# B&R Automation Studio project NAEUL004C00R13L518F00 (part 18)

#### Act_OptP0929MagConv2BtmDC.st
```iecst
ACTION Act_OptP0929MagConv2BtmDC:

	//Magazine Conv2eyor
	IF tyP0929MagConv2.tyBtmDC.tyBtnStop.bRtCompl = TRUE THEN
		eOutMagConv2Act	:= MagConvActStop;

		IF p_eOutMagConv2Stat = MagConvActStop AND p_eOutMagConv2Status = Done THEN
			eOutMagConv2Act	:= MagConvActIdle;

			tyP0929MagConv2.tyBtmDC.tyBtnStop.bRtCompl		:= FALSE;
			tyP0929MagConv2.tyBtmDC.tyBtnStop.bValue		:= TRUE;
			tyP0929MagConv2.tyBtmDC.tyBtnStop.bRtLk		:= TRUE;

			tyP0929MagConv2.tyBtmDC.tyBtnMagIn.bRtCompl	:= FALSE;
			tyP0929MagConv2.tyBtmDC.tyBtnMagIn.bValue		:= FALSE;
			tyP0929MagConv2.tyBtmDC.tyBtnMagIn.bRtLk		:= FALSE;

			tyP0929MagConv2.tyBtmDC.tyBtnMagOut.bRtCompl	:= FALSE;
			tyP0929MagConv2.tyBtmDC.tyBtnMagOut.bValue		:= FALSE;
			tyP0929MagConv2.tyBtmDC.tyBtnMagOut.bRtLk		:= FALSE;
		END_IF

	ELSIF tyP0929MagConv2.tyBtmDC.tyBtnMagIn.bRtCompl = TRUE THEN
		tyP0929MagConv2.tyBtmDC.tyBtnMagIn.bValue	:= TRUE;
		tyP0929MagConv2.tyBtmDC.tyBtnMagIn.bRtLk	:= TRUE;

		tyP0929MagConv2.tyBtmDC.tyBtnStop.bValue	:= FALSE;
		tyP0929MagConv2.tyBtmDC.tyBtnStop.bRtLk	:= FALSE;

		IF p_tyNtParamCurr.eProjOutMagConv2Dir = ConvDirLToR OR p_tyNtParamCurr.eProjOutMagConv2Dir = ConvDirLToL THEN

			eOutMagConv2Act	:= MagConvActSetMtrSigOnOrLToR;

			IF p_eOutMagConv2Stat = MagConvActSetMtrSigOnOrLToR AND p_eOutMagConv2Status = Done THEN
				eOutMagConv2Act	:= MagConvActIdle;

				tyP0929MagConv2.tyBtmDC.tyBtnMagIn.bRtCompl	:= FALSE;
			END_IF

		ELSE

			eOutMagConv2Act	:= MagConvActSetMtrDirOrRToL;

			IF p_eOutMagConv2Stat = MagConvActSetMtrDirOrRToL AND p_eOutMagConv2Status = Done THEN
				eOutMagConv2Act	:= MagConvActIdle;

				tyP0929MagConv2.tyBtmDC.tyBtnMagIn.bRtCompl	:= FALSE;
			END_IF

		END_IF

	ELSIF tyP0929MagConv2.tyBtmDC.tyBtnMagOut.bRtCompl = TRUE THEN
		tyP0929MagConv2.tyBtmDC.tyBtnMagOut.bValue	:= TRUE;
		tyP0929MagConv2.tyBtmDC.tyBtnMagOut.bRtLk	:= TRUE;

		tyP0929MagConv2.tyBtmDC.tyBtnStop.bValue	:= FALSE;
		tyP0929MagConv2.tyBtmDC.tyBtnStop.bRtLk	:= FALSE;

		IF p_tyNtParamCurr.eProjOutMagConv2Dir = ConvDirLToR OR p_tyNtParamCurr.eProjOutMagConv2Dir = ConvDirRToR THEN

			eOutMagConv2Act	:= MagConvActSetMtrSigOnOrLToR;

			IF p_eOutMagConv2Stat = MagConvActSetMtrSigOnOrLToR AND p_eOutMagConv2Status = Done THEN
				eOutMagConv2Act	:= MagConvActIdle;

				tyP0929MagConv2.tyBtmDC.tyBtnMagOut.bRtCompl	:= FALSE;
			END_IF

		ELSE

			eOutMagConv2Act	:= MagConvActSetMtrDirOrRToL;

			IF p_eOutMagConv2Stat = MagConvActSetMtrDirOrRToL AND p_eOutMagConv2Status = Done THEN
				eOutMagConv2Act	:= MagConvActIdle;

				tyP0929MagConv2.tyBtmDC.tyBtnMagOut.bRtCompl	:= FALSE;
			END_IF

		END_IF

	END_IF

	IF tyP0929MagConv2.tyCom.tyBtnSwitch.bValue = TRUE THEN

		//Mag Conv2 Stopper4
		IF p_bStopper4TwoCtrlOut = FALSE THEN
			IF tyP0929MagConv2.tyBtmDC.tyBtnMidStprExt.bRtCompl = TRUE THEN
				tyP0929MagConv2.tyBtmDC.tyBtnMidStprExt.bValue := TRUE;
				tyP0929MagConv2.tyBtmDC.tyBtnMidStprRet.bValue := FALSE;

				eStopper4Act2	:= PneuActSetExt;

				IF p_eStopper4Stat2 = PneuActSetExt AND p_eStopper4Status2 = Done THEN
					eStopper4Act2	:= PneuActIdle;

					tyP0929MagConv2.tyBtmDC.tyBtnMidStprExt.bRtCompl	:= FALSE;
				END_IF

			ELSIF tyP0929MagConv2.tyBtmDC.tyBtnMidStprRet.bRtCompl = TRUE THEN
				tyP0929MagConv2.tyBtmDC.tyBtnMidStprRet.bValue := TRUE;
				tyP0929MagConv2.tyBtmDC.tyBtnMidStprExt.bValue := FALSE;

				eStopper4Act2	:= PneuActSetRet;

				IF p_eStopper4Stat2 = PneuActSetRet AND p_eStopper4Status2 = Done THEN
					eStopper4Act2	:= PneuActIdle;

					tyP0929MagConv2.tyBtmDC.tyBtnMidStprRet.bRtCompl	:= FALSE;
				END_IF
			END_IF

		ELSE
			IF (tyP0929MagConv2.tyBtmDC.tyBtnMidStprExt.bRtCompl = TRUE) OR (tyP0929MagConv2.tyBtmDC.tyBtnMidStprRet.bRtCompl = TRUE) THEN
				IF (tyP0929MagConv2.tyBtmDC.tyBtnMidStprExt.bValue = TRUE) AND (tyP0929MagConv2.tyBtmDC.tyBtnMidStprRet.bValue = TRUE) THEN
					eStopper4Act2	:= PneuActSetAll;

					IF p_eStopper4Stat2 = PneuActSetAll AND p_eStopper4Status2 = Done THEN
						eStopper4Act2	:= PneuActIdle;

						tyP0929MagConv2.tyBtmDC.tyBtnMidStprExt.bRtCompl		:= FALSE;
						tyP0929MagConv2.tyBtmDC.tyBtnMidStprRet.bRtCompl			:= FALSE;
					END_IF
					/////////i edited the ret to ext
				ELSIF (tyP0929MagConv2.tyBtmDC.tyBtnMidStprExt.bValue = TRUE) AND (tyP0929MagConv2.tyBtmDC.tyBtnMidStprRet.bValue = FALSE) THEN
					eStopper4Act2	:= PneuActSetExt;(**)

					IF p_eStopper4Stat2 = PneuActSetExt (**) AND p_eStopper4Status2 = Done THEN
						eStopper4Act2	:= PneuActIdle;

						tyP0929MagConv2.tyBtmDC.tyBtnMidStprExt.bRtCompl		:= FALSE;
						tyP0929MagConv2.tyBtmDC.tyBtnMidStprRet.bRtCompl		:= FALSE;
					END_IF

				ELSIF (tyP0929MagConv2.tyBtmDC.tyBtnMidStprExt.bValue = FALSE) AND (tyP0929MagConv2.tyBtmDC.tyBtnMidStprRet.bValue = TRUE) THEN
					eStopper4Act2	:= PneuActSetRet;

					IF p_eStopper4Stat2 = PneuActSetRet AND p_eStopper4Status2 = Done THEN
						eStopper4Act2	:= PneuActIdle;

						tyP0929MagConv2.tyBtmDC.tyBtnMidStprExt.bRtCompl		:= FALSE;
						tyP0929MagConv2.tyBtmDC.tyBtnMidStprRet.bRtCompl			:= FALSE;
					END_IF
					///////
				ELSE
					eStopper4Act2	:= PneuActRstAll;

					IF p_eStopper4Stat2 = PneuActRstAll AND p_eStopper4Status2 = Done THEN
						eStopper4Act2	:= PneuActIdle;

						tyP0929MagConv2.tyBtmDC.tyBtnMidStprExt.bRtCompl		:= FALSE;
						tyP0929MagConv2.tyBtmDC.tyBtnMidStprRet.bRtCompl			:= FALSE;
					END_IF

				END_IF
			END_IF
		END_IF//Stopper4

		//Mag Conv2 Stopper5
		IF p_bStopper5TwoCtrlOut = FALSE THEN
			IF tyP0929MagConv2.tyBtmDC.tyBtnExtStprExt.bRtCompl = TRUE THEN
				tyP0929MagConv2.tyBtmDC.tyBtnExtStprExt.bValue := TRUE;
				tyP0929MagConv2.tyBtmDC.tyBtnExtStprRet.bValue := FALSE;

				eStopper5Act2	:= PneuActSetExt;

				IF p_eStopper5Stat2 = PneuActSetExt AND p_eStopper5Status2 = Done THEN
					eStopper5Act2	:= PneuActIdle;

					tyP0929MagConv2.tyBtmDC.tyBtnExtStprExt.bRtCompl	:= FALSE;
				END_IF

			ELSIF tyP0929MagConv2.tyBtmDC.tyBtnExtStprRet.bRtCompl = TRUE THEN
				tyP0929MagConv2.tyBtmDC.tyBtnExtStprRet.bValue := TRUE;
				tyP0929MagConv2.tyBtmDC.tyBtnExtStprExt.bValue := FALSE;

				eStopper5Act2	:= PneuActSetRet;

				IF p_eStopper5Stat2 = PneuActSetRet AND p_eStopper5Status2 = Done THEN
					eStopper5Act2	:= PneuActIdle;

					tyP0929MagConv2.tyBtmDC.tyBtnExtStprRet.bRtCompl	:= FALSE;
				END_IF
			END_IF

		ELSE
			IF (tyP0929MagConv2.tyBtmDC.tyBtnExtStprExt.bRtCompl = TRUE) OR (tyP0929MagConv2.tyBtmDC.tyBtnExtStprRet.bRtCompl = TRUE) THEN
				IF (tyP0929MagConv2.tyBtmDC.tyBtnExtStprExt.bValue = TRUE) AND (tyP0929MagConv2.tyBtmDC.tyBtnExtStprRet.bValue = TRUE) THEN
					eStopper5Act2	:= PneuActSetAll;

					IF p_eStopper5Stat2 = PneuActSetAll AND p_eStopper5Status2 = Done THEN
						eStopper5Act2	:= PneuActIdle;

						tyP0929MagConv2.tyBtmDC.tyBtnExtStprExt.bRtCompl		:= FALSE;
						tyP0929MagConv2.tyBtmDC.tyBtnExtStprRet.bRtCompl			:= FALSE;
					END_IF
					/////////i edited the ret to ext
				ELSIF (tyP0929MagConv2.tyBtmDC.tyBtnExtStprExt.bValue = TRUE) AND (tyP0929MagConv2.tyBtmDC.tyBtnExtStprRet.bValue = FALSE) THEN
					eStopper5Act2	:= PneuActSetExt;(**)

					IF p_eStopper5Stat2 = PneuActSetExt (**) AND p_eStopper5Status2 = Done THEN
						eStopper5Act2	:= PneuActIdle;

						tyP0929MagConv2.tyBtmDC.tyBtnExtStprExt.bRtCompl		:= FALSE;
						tyP0929MagConv2.tyBtmDC.tyBtnExtStprRet.bRtCompl		:= FALSE;
					END_IF

				ELSIF (tyP0929MagConv2.tyBtmDC.tyBtnExtStprExt.bValue = FALSE) AND (tyP0929MagConv2.tyBtmDC.tyBtnExtStprRet.bValue = TRUE) THEN
					eStopper5Act2	:= PneuActSetRet;

					IF p_eStopper5Stat2 = PneuActSetRet AND p_eStopper5Status2 = Done THEN
						eStopper5Act2	:= PneuActIdle;

						tyP0929MagConv2.tyBtmDC.tyBtnExtStprExt.bRtCompl		:= FALSE;
						tyP0929MagConv2.tyBtmDC.tyBtnExtStprRet.bRtCompl			:= FALSE;
					END_IF
					///////
				ELSE
					eStopper5Act2	:= PneuActRstAll;

					IF p_eStopper5Stat2 = PneuActRstAll AND p_eStopper5Status2 = Done THEN
						eStopper5Act2	:= PneuActIdle;

						tyP0929MagConv2.tyBtmDC.tyBtnExtStprExt.bRtCompl		:= FALSE;
						tyP0929MagConv2.tyBtmDC.tyBtnExtStprRet.bRtCompl			:= FALSE;
					END_IF

				END_IF
			END_IF
		END_IF//Stopper5

		//mid
		tyP0929MagConv2.tyBtmFB.tyBtnMidStprExt.bRtCompl		:= FALSE;
		tyP0929MagConv2.tyBtmFB.tyBtnMidStprExt.bValue		:= FALSE;
		tyP0929MagConv2.tyBtmFB.tyBtnMidStprRet.bRtCompl		:= FALSE;
		tyP0929MagConv2.tyBtmFB.tyBtnMidStprRet.bValue		:= FALSE;

		//ext
		tyP0929MagConv2.tyBtmFB.tyBtnExtStprExt.bRtCompl		:= FALSE;
		tyP0929MagConv2.tyBtmFB.tyBtnExtStprExt.bValue		:= FALSE;
		tyP0929MagConv2.tyBtmFB.tyBtnExtStprRet.bRtCompl		:= FALSE;
		tyP0929MagConv2.tyBtmFB.tyBtnExtStprRet.bValue		:= FALSE;
	END_IF

	//Mask
//	IF p_eOutMagConv2Status = Error THEN
//
//		fUIInRtStatOff(ADR(tyP0929MagConv2.tyBtmDC.tyBtnMagIn.uiMaskRtStat));
//		fUIInRtStatOff(ADR(tyP0929MagConv2.tyBtmDC.tyBtnMagOut.uiMaskRtStat));
//		fUIInRtStatOff(ADR(tyP0929MagConv2.tyBtmDC.tyBtnFixedClamp.uiMaskRtStat));
//		fUIInRtStatOff(ADR(tyP0929MagConv2.tyBtmDC.tyBtnFixedUnclamp.uiMaskRtStat));
//		fUIInRtStatOff(ADR(tyP0929MagConv2.tyBtmDC.tyBtnRemoteClamp.uiMaskRtStat));
//		fUIInRtStatOff(ADR(tyP0929MagConv2.tyBtmDC.tyBtnRemoteUnclamp.uiMaskRtStat));
//		fUIInRtStatOff(ADR(tyP0929MagConv2.tyBtmDC.tyBtnSelClamp.uiMaskRtStat));
//		fUIInRtStatOff(ADR(tyP0929MagConv2.tyBtmDC.tyBtnSelUnclamp.uiMaskRtStat));
//
//	ELSIF tyP0929MagConv2.tyBtmDC.tyBtnMagIn.bValue = TRUE THEN
//
//		fUIInRtStatHide(ADR(tyP0929MagConv2.tyBtmDC.tyBtnMagIn.uiMaskRtStat));
//		fUIInRtStatOff(ADR(tyP0929MagConv2.tyBtmDC.tyBtnMagOut.uiMaskRtStat));
//		fUIInRtStatOff(ADR(tyP0929MagConv2.tyBtmDC.tyBtnFixedClamp.uiMaskRtStat));
//		fUIInRtStatOff(ADR(tyP0929MagConv2.tyBtmDC.tyBtnFixedUnclamp.uiMaskRtStat));
//		fUIInRtStatOff(ADR(tyP0929MagConv2.tyBtmDC.tyBtnRemoteClamp.uiMaskRtStat));
//		fUIInRtStatOff(ADR(tyP0929MagConv2.tyBtmDC.tyBtnRemoteUnclamp.uiMaskRtStat));
//		fUIInRtStatOff(ADR(tyP0929MagConv2.tyBtmDC.tyBtnSelClamp.uiMaskRtStat));
//		fUIInRtStatOff(ADR(tyP0929MagConv2.tyBtmDC.tyBtnSelUnclamp.uiMaskRtStat));
//
//	ELSIF tyP0929MagConv2.tyBtmDC.tyBtnMagOut.bValue = TRUE THEN
//
//		fUIInRtStatOff(ADR(tyP0929MagConv2.tyBtmDC.tyBtnMagIn.uiMaskRtStat));
//		fUIInRtStatHide(ADR(tyP0929MagConv2.tyBtmDC.tyBtnMagOut.uiMaskRtStat));
//		fUIInRtStatOff(ADR(tyP0929MagConv2.tyBtmDC.tyBtnFixedClamp.uiMaskRtStat));
//		fUIInRtStatOff(ADR(tyP0929MagConv2.tyBtmDC.tyBtnFixedUnclamp.uiMaskRtStat));
//		fUIInRtStatOff(ADR(tyP0929MagConv2.tyBtmDC.tyBtnRemoteClamp.uiMaskRtStat));
//		fUIInRtStatOff(ADR(tyP0929MagConv2.tyBtmDC.tyBtnRemoteUnclamp.uiMaskRtStat));
//		fUIInRtStatOff(ADR(tyP0929MagConv2.tyBtmDC.tyBtnSelClamp.uiMaskRtStat));
//		fUIInRtStatOff(ADR(tyP0929MagConv2.tyBtmDC.tyBtnSelUnclamp.uiMaskRtStat));
//
//	ELSE
//
//		fUIInRtStatHide(ADR(tyP0929MagConv2.tyBtmDC.tyBtnMagIn.uiMaskRtStat));
//		fUIInRtStatHide(ADR(tyP0929MagConv2.tyBtmDC.tyBtnMagOut.uiMaskRtStat));
//		fUIInRtStatHide(ADR(tyP0929MagConv2.tyBtmDC.tyBtnFixedClamp.uiMaskRtStat));
//		fUIInRtStatHide(ADR(tyP0929MagConv2.tyBtmDC.tyBtnFixedUnclamp.uiMaskRtStat));
//		fUIInRtStatHide(ADR(tyP0929MagConv2.tyBtmDC.tyBtnRemoteClamp.uiMaskRtStat));
//		fUIInRtStatHide(ADR(tyP0929MagConv2.tyBtmDC.tyBtnRemoteUnclamp.uiMaskRtStat));
//		fUIInRtStatHide(ADR(tyP0929MagConv2.tyBtmDC.tyBtnSelClamp.uiMaskRtStat));
//		fUIInRtStatHide(ADR(tyP0929MagConv2.tyBtmDC.tyBtnSelUnclamp.uiMaskRtStat));
//
//	END_IF
//

END_ACTION
```

#### Act_OptP0929RstMnlTop.st
```iecst
ACTION Act_OptP0929RstMnlTop:

	IF EDGEPOS((bManualMod = FALSE) OR (p_eInMagConv2Status = Error)) THEN

		eInMagConv2Act	:= MagConvActIdle;
		//Magazine Conv2eyor
		//FB
		tyP0929MagConv2.tyTopFB.tyBtnEnt.bRtCompl				:= FALSE;
		tyP0929MagConv2.tyTopFB.tyBtnExit.bRtCompl				:= FALSE;
		tyP0929MagConv2.tyTopFB.tyBtnStop.bRtCompl				:= FALSE;

		tyP0929MagConv2.tyTopFB.tyBtnEnt.bValue				:= FALSE;
		tyP0929MagConv2.tyTopFB.tyBtnExit.bValue				:= FALSE;
		tyP0929MagConv2.tyTopFB.tyBtnStop.bValue				:= TRUE;

		tyP0929MagConv2.tyTopFB.tyBtnEnt.bRtLk				:= FALSE;
		tyP0929MagConv2.tyTopFB.tyBtnExit.bRtLk				:= FALSE;
		tyP0929MagConv2.tyTopFB.tyBtnStop.bRtLk				:= TRUE;

		tyP0929MagConv2.tyTopFB.tyBtnEnt.uiMaskRtStat.0		:= TRUE;
		tyP0929MagConv2.tyTopFB.tyBtnExit.uiMaskRtStat.0		:= TRUE;
		tyP0929MagConv2.tyCom.tyBtnSwitch.uiMaskRtStat.0		:= TRUE;

		//Direct
		tyP0929MagConv2.tyTopDC.tyBtnMagIn.bRtCompl				:= FALSE;
		tyP0929MagConv2.tyTopDC.tyBtnMagOut.bRtCompl				:= FALSE;
		tyP0929MagConv2.tyTopDC.tyBtnStop.bRtCompl				:= FALSE;

		tyP0929MagConv2.tyTopDC.tyBtnMagIn.bValue				:= FALSE;
		tyP0929MagConv2.tyTopDC.tyBtnMagOut.bValue				:= FALSE;
		tyP0929MagConv2.tyTopDC.tyBtnStop.bValue					:= TRUE;

		tyP0929MagConv2.tyTopDC.tyBtnMagIn.bRtLk					:= FALSE;
		tyP0929MagConv2.tyTopDC.tyBtnMagOut.bRtLk				:= FALSE;
		tyP0929MagConv2.tyTopDC.tyBtnStop.bRtLk					:= TRUE;

		tyP0929MagConv2.tyTopDC.tyBtnMagIn.uiMaskRtStat.0		:= TRUE;
		tyP0929MagConv2.tyTopDC.tyBtnMagOut.uiMaskRtStat.0		:= TRUE;
		tyP0929MagConv2.tyCom.tyBtnSwitch.uiMaskRtStat.0			:= TRUE;

		//Magazine Clamper
		//FB
		//Top
		tyP0929MagConv2.tyTopFB.tyBtnEntStprExt.bRtCompl			:= FALSE;
		tyP0929MagConv2.tyTopFB.tyBtnEntStprRet.bRtCompl			:= FALSE;

		tyP0929MagConv2.tyTopFB.tyBtnEntStprExt.bValue				:= FALSE;
		tyP0929MagConv2.tyTopFB.tyBtnEntStprRet.bValue			:= FALSE;

		//Remote
		tyP0929MagConv2.tyTopFB.tyBtnMidStprExt.bRtCompl			:= FALSE;
		tyP0929MagConv2.tyTopFB.tyBtnMidStprRet.bRtCompl		:= FALSE;

		tyP0929MagConv2.tyTopFB.tyBtnMidStprExt.bValue			:= FALSE;
		tyP0929MagConv2.tyTopFB.tyBtnMidStprRet.bValue			:= FALSE;

		//Top
		tyP0929MagConv2.tyTopFB.tyBtnExtStprExt.bRtCompl			:= FALSE;
		tyP0929MagConv2.tyTopFB.tyBtnExtStprRet.bRtCompl		:= FALSE;

		tyP0929MagConv2.tyTopFB.tyBtnExtStprExt.bValue			:= FALSE;
		tyP0929MagConv2.tyTopFB.tyBtnExtStprRet.bValue			:= FALSE;

		tyP0929MagConv2.tyTopFB.tyBtnEntStprExt.uiMaskRtStat.0		:= TRUE;
		tyP0929MagConv2.tyTopFB.tyBtnEntStprRet.uiMaskRtStat.0	:= TRUE;
		tyP0929MagConv2.tyTopFB.tyBtnMidStprExt.uiMaskRtStat.0	:= TRUE;
		tyP0929MagConv2.tyTopFB.tyBtnMidStprRet.uiMaskRtStat.0	:= TRUE;
		tyP0929MagConv2.tyTopFB.tyBtnExtStprExt.uiMaskRtStat.0		:= TRUE;
		tyP0929MagConv2.tyTopFB.tyBtnExtStprRet.uiMaskRtStat.0		:= TRUE;

		tyP0929MagConv2.tyCom.tyBtnSwitch.uiMaskRtStat.0		:= TRUE;

		//Direct
		//Fixed
		tyP0929MagConv2.tyTopDC.tyBtnEntStprExt.bRtCompl			:= FALSE;
		tyP0929MagConv2.tyTopDC.tyBtnEntStprRet.bRtCompl			:= FALSE;

		tyP0929MagConv2.tyTopDC.tyBtnEntStprExt.bValue				:= FALSE;
		tyP0929MagConv2.tyTopDC.tyBtnEntStprRet.bValue			:= FALSE;

		//Remote
		tyP0929MagConv2.tyTopDC.tyBtnMidStprExt.bRtCompl			:= FALSE;
		tyP0929MagConv2.tyTopDC.tyBtnMidStprRet.bRtCompl		:= FALSE;

		tyP0929MagConv2.tyTopDC.tyBtnMidStprExt.bValue			:= FALSE;
		tyP0929MagConv2.tyTopDC.tyBtnMidStprRet.bValue			:= FALSE;

		//Top
		tyP0929MagConv2.tyTopDC.tyBtnExtStprExt.bRtCompl				:= FALSE;
		tyP0929MagConv2.tyTopDC.tyBtnExtStprRet.bRtCompl			:= FALSE;

		tyP0929MagConv2.tyTopDC.tyBtnExtStprExt.bValue				:= FALSE;
		tyP0929MagConv2.tyTopDC.tyBtnExtStprRet.bValue				:= FALSE;

		tyP0929MagConv2.tyTopDC.tyBtnEntStprExt.uiMaskRtStat.0		:= TRUE;
		tyP0929MagConv2.tyTopDC.tyBtnEntStprRet.uiMaskRtStat.0	:= TRUE;
		tyP0929MagConv2.tyTopDC.tyBtnMidStprExt.uiMaskRtStat.0	:= TRUE;
		tyP0929MagConv2.tyTopDC.tyBtnMidStprRet.uiMaskRtStat.0	:= TRUE;
		tyP0929MagConv2.tyTopDC.tyBtnExtStprExt.uiMaskRtStat.0		:= TRUE;
		tyP0929MagConv2.tyTopDC.tyBtnExtStprRet.uiMaskRtStat.0		:= TRUE;

		tyP0929MagConv2.tyCom.tyBtnSwitch.uiMaskRtStat.0		:= TRUE;

	END_IF

END_ACTION
```

#### Act_OptP0929RstMnlBtm.st
```iecst
ACTION Act_OptP0929RstMnlBtm:

	IF EDGEPOS((bManualMod = FALSE) OR (p_eOutMagConv2Status = Error)) THEN

		eOutMagConv2Act	:= MagConvActIdle;
		//Magazine Conv2eyor
		//FB
		tyP0929MagConv2.tyBtmFB.tyBtnEnt.bRtCompl				:= FALSE;
		tyP0929MagConv2.tyBtmFB.tyBtnExit.bRtCompl				:= FALSE;
		tyP0929MagConv2.tyBtmFB.tyBtnStop.bRtCompl				:= FALSE;

		tyP0929MagConv2.tyBtmFB.tyBtnEnt.bValue				:= FALSE;
		tyP0929MagConv2.tyBtmFB.tyBtnExit.bValue				:= FALSE;
		tyP0929MagConv2.tyBtmFB.tyBtnStop.bValue				:= TRUE;

		tyP0929MagConv2.tyBtmFB.tyBtnEnt.bRtLk				:= FALSE;
		tyP0929MagConv2.tyBtmFB.tyBtnExit.bRtLk				:= FALSE;
		tyP0929MagConv2.tyBtmFB.tyBtnStop.bRtLk				:= TRUE;

		tyP0929MagConv2.tyBtmFB.tyBtnEnt.uiMaskRtStat.0		:= TRUE;
		tyP0929MagConv2.tyBtmFB.tyBtnExit.uiMaskRtStat.0		:= TRUE;
		tyP0929MagConv2.tyCom.tyBtnSwitch.uiMaskRtStat.0		:= TRUE;

		//Direct
		tyP0929MagConv2.tyBtmDC.tyBtnMagIn.bRtCompl				:= FALSE;
		tyP0929MagConv2.tyBtmDC.tyBtnMagOut.bRtCompl				:= FALSE;
		tyP0929MagConv2.tyBtmDC.tyBtnStop.bRtCompl				:= FALSE;

		tyP0929MagConv2.tyBtmDC.tyBtnMagIn.bValue				:= FALSE;
		tyP0929MagConv2.tyBtmDC.tyBtnMagOut.bValue				:= FALSE;
		tyP0929MagConv2.tyBtmDC.tyBtnStop.bValue					:= TRUE;

		tyP0929MagConv2.tyBtmDC.tyBtnMagIn.bRtLk					:= FALSE;
		tyP0929MagConv2.tyBtmDC.tyBtnMagOut.bRtLk				:= FALSE;
		tyP0929MagConv2.tyBtmDC.tyBtnStop.bRtLk					:= TRUE;

		tyP0929MagConv2.tyBtmDC.tyBtnMagIn.uiMaskRtStat.0		:= TRUE;
		tyP0929MagConv2.tyBtmDC.tyBtnMagOut.uiMaskRtStat.0		:= TRUE;
		tyP0929MagConv2.tyCom.tyBtnSwitch.uiMaskRtStat.0			:= TRUE;

		//Magazine Clamper
		//FB
		//Remote
		tyP0929MagConv2.tyBtmFB.tyBtnMidStprExt.bRtCompl			:= FALSE;
		tyP0929MagConv2.tyBtmFB.tyBtnMidStprRet.bRtCompl		:= FALSE;

		tyP0929MagConv2.tyBtmFB.tyBtnMidStprExt.bValue			:= FALSE;
		tyP0929MagConv2.tyBtmFB.tyBtnMidStprRet.bValue			:= FALSE;

		//Top
		tyP0929MagConv2.tyBtmFB.tyBtnExtStprExt.bRtCompl			:= FALSE;
		tyP0929MagConv2.tyBtmFB.tyBtnExtStprRet.bRtCompl		:= FALSE;

		tyP0929MagConv2.tyBtmFB.tyBtnExtStprExt.bValue			:= FALSE;
		tyP0929MagConv2.tyBtmFB.tyBtnExtStprRet.bValue			:= FALSE;

		tyP0929MagConv2.tyBtmFB.tyBtnMidStprExt.uiMaskRtStat.0	:= TRUE;
		tyP0929MagConv2.tyBtmFB.tyBtnMidStprRet.uiMaskRtStat.0	:= TRUE;
		tyP0929MagConv2.tyBtmFB.tyBtnExtStprExt.uiMaskRtStat.0		:= TRUE;
		tyP0929MagConv2.tyBtmFB.tyBtnExtStprRet.uiMaskRtStat.0		:= TRUE;

		tyP0929MagConv2.tyCom.tyBtnSwitch.uiMaskRtStat.0		:= TRUE;

		//Direct
		//Fixed

		//Remote
		tyP0929MagConv2.tyBtmDC.tyBtnMidStprExt.bRtCompl			:= FALSE;
		tyP0929MagConv2.tyBtmDC.tyBtnMidStprRet.bRtCompl		:= FALSE;

		tyP0929MagConv2.tyBtmDC.tyBtnMidStprExt.bValue			:= FALSE;
		tyP0929MagConv2.tyBtmDC.tyBtnMidStprRet.bValue			:= FALSE;

		//Top
		tyP0929MagConv2.tyBtmDC.tyBtnExtStprExt.bRtCompl				:= FALSE;
		tyP0929MagConv2.tyBtmDC.tyBtnExtStprRet.bRtCompl			:= FALSE;

		tyP0929MagConv2.tyBtmDC.tyBtnExtStprExt.bValue				:= FALSE;
		tyP0929MagConv2.tyBtmDC.tyBtnExtStprRet.bValue				:= FALSE;

		tyP0929MagConv2.tyBtmDC.tyBtnMidStprExt.uiMaskRtStat.0	:= TRUE;
		tyP0929MagConv2.tyBtmDC.tyBtnMidStprRet.uiMaskRtStat.0	:= TRUE;
		tyP0929MagConv2.tyBtmDC.tyBtnExtStprExt.uiMaskRtStat.0		:= TRUE;
		tyP0929MagConv2.tyBtmDC.tyBtnExtStprRet.uiMaskRtStat.0		:= TRUE;

		tyP0929MagConv2.tyCom.tyBtnSwitch.uiMaskRtStat.0		:= TRUE;

	END_IF

END_ACTION
```

#### Act_EntP0930Disp.st
```iecst
ACTION Act_EntP0930Disp:

	//Access Address
	p_tyC0002FullMask ACCESS ADR(tyP0930MagConv1.tyFullMaskHide);

	//p_tyC0004Navi ACCESS ADR(tyP0930MagConv1.tyNaviBack);

	CASE p_tyNtParamCurr.eProjMag OF
		ULMagDual:
			p_tyC0004Navi ACCESS ADR(tyP0930MagConv1.tyNavi2Lyr1);
		ULMagTriple:
			p_tyC0004Navi ACCESS ADR(tyP0930MagConv1.tyNavi3Lyr1);
	END_CASE

	p_tyC0005Main ACCESS ADR(tyCommon.tyMain);

	p_tyC0007Notif ACCESS ADR(tyCommon.tyNotif);

	p_tyC0008MsgBox ACCESS ADR(tyP0930MagConv1.tyMsgBoxHide);

	p_tyC0009Info ACCESS ADR(tyCommon.tyInfo);

	p_tyP0930Mag1ConvCom ACCESS ADR(tyP0930MagConv1.tyCom);
	p_tyP0930Mag1ConvDC ACCESS ADR(tyP0930MagConv1.tyDC);
	p_tyP0930Mag1ConvFB ACCESS ADR(tyP0930MagConv1.tyFB);

	IF p_tyNtParamCurr.bMagAutoVerifyPrep AND p_tyNtParamCurr.bProjMagAWPrep THEN
		IF p_tyNtParamCurr.eProjMag = ULMagDual THEN
			tyP0930MagConv1.tyCom.tyBitmapMc.uiValueIdx	:= 103;
		END_IF
	ELSIF p_tyNtParamCurr.bMagAutoVerifyPrep = FALSE AND p_tyNtParamCurr.bProjMagAWPrep = FALSE THEN
		IF p_tyNtParamCurr.eProjMag = ULMagDual THEN
			tyP0930MagConv1.tyCom.tyBitmapMc.uiValueIdx	:= 105;
		END_IF
	ELSE
		tyP0930MagConv1.tyCom.tyBitmapMc.uiValueIdx	:= 233;
	END_IF

	tyP0930MagConv1.tyFullMaskAWMotorEngage.tyBtnMask.bRtLk			:=FALSE;

	IF p_tyNtParamCurr.bMagAutoVerifyPrep = FALSE THEN
		IF tyP0930MagConv1.tyCom.tyBtnSwitch.bValue THEN
			fUIInRtStatHide(ADR(tyP0930MagConv1.tyFB.tyLyr.uiRtStat));
			fUIInRtStatHide(ADR(tyP0930MagConv1.tyDC.tyLyr.uiRtStat));
			fUIInRtStatHide(ADR(tyP0930MagConv1.tyFB.tyLyrWithoutSelClamp.uiRtStat));
			fUIInRtStatOff(ADR(tyP0930MagConv1.tyDC.tyLyrWithoutSelClamp.uiRtStat));
		ELSE
			fUIInRtStatHide(ADR(tyP0930MagConv1.tyFB.tyLyr.uiRtStat));
			fUIInRtStatHide(ADR(tyP0930MagConv1.tyDC.tyLyr.uiRtStat));
			fUIInRtStatOff(ADR(tyP0930MagConv1.tyFB.tyLyrWithoutSelClamp.uiRtStat));
			fUIInRtStatHide(ADR(tyP0930MagConv1.tyDC.tyLyrWithoutSelClamp.uiRtStat));
		END_IF
	ELSE
		IF tyP0930MagConv1.tyCom.tyBtnSwitch.bValue THEN
			fUIInRtStatHide(ADR(tyP0930MagConv1.tyFB.tyLyr.uiRtStat));
			fUIInRtStatOff(ADR(tyP0930MagConv1.tyDC.tyLyr.uiRtStat));
			fUIInRtStatHide(ADR(tyP0930MagConv1.tyFB.tyLyrWithoutSelClamp.uiRtStat));
			fUIInRtStatHide(ADR(tyP0930MagConv1.tyDC.tyLyrWithoutSelClamp.uiRtStat));
		ELSE
			fUIInRtStatOff(ADR(tyP0930MagConv1.tyFB.tyLyr.uiRtStat));
			fUIInRtStatHide(ADR(tyP0930MagConv1.tyDC.tyLyr.uiRtStat));
			fUIInRtStatHide(ADR(tyP0930MagConv1.tyFB.tyLyrWithoutSelClamp.uiRtStat));
			fUIInRtStatHide(ADR(tyP0930MagConv1.tyDC.tyLyrWithoutSelClamp.uiRtStat));
		END_IF
	END_IF
END_ACTION
```

#### Act_OptP0930FullMask.st
```iecst
ACTION Act_OptP0930FullMask:

	IF eCurrPage = UIP0930MagConv1 THEN

		IF p_tyDI.bEStopSig = FALSE THEN
			p_tyC0002FullMask ACCESS ADR(tyP0930MagConv1.tyFullMaskEStop);

		ELSIF p_tyDI.bCoverSWSig = FALSE THEN
			p_tyC0002FullMask ACCESS ADR(tyP0930MagConv1.tyFullMaskCWSig);

		ELSIF p_tyDI.bSafetyRlySig = FALSE THEN
			p_tyC0002FullMask ACCESS ADR(tyP0930MagConv1.tyFullMaskSafetyRly);

		ELSIF p_bMag1AWEngageExtCtrl
			AND NOT p_bMagConv2Clp1ClprFixClampCtrl
			AND NOT p_bMagConv2Clp1ClprRmtClampCtrl
			THEN
			p_tyC0002FullMask ACCESS ADR(tyP0930MagConv1.tyFullMaskAWMotorEngage);

		ELSE
			p_tyC0002FullMask ACCESS ADR(tyP0930MagConv1.tyFullMaskHide);

		END_IF

	END_IF

END_ACTION
```

#### Act_OptP0930Navi.st
```iecst
ACTION Act_OptP0930Navi:

//	IF tyP0930MagConv1.tyNaviBack.tyBtnBack.bRtCompl = TRUE THEN
//		tyP0930MagConv1.tyNaviBack.tyBtnBack.bRtCompl	:= FALSE;
//		tyP0930MagConv1.tyNaviBack.tyBtnBack.bValue		:= FALSE;
//
//		eChgPage	:= UIP0920MtrNPneuCtrl;
//	END_IF

	CASE p_tyNtParamCurr.eProjMag OF
		ULMagDual:
			IF tyP0930MagConv1.tyNavi2Lyr1.tyBtnBack.bRtCompl = TRUE THEN
				tyP0930MagConv1.tyNavi2Lyr1.tyBtnBack.bRtCompl	:= FALSE;
				tyP0930MagConv1.tyNavi2Lyr1.tyBtnBack.bValue		:= FALSE;

				eChgPage	:= UIP0920MtrNPneuCtrl;
				bDispMagConv1	:= TRUE;
				bDispMagConv2	:= FALSE;
				bDispMagConv3	:= FALSE;

			ELSIF tyP0930MagConv1.tyNavi2Lyr1.tyBtnLeft.bRtCompl = TRUE OR tyP0930MagConv1.tyNavi2Lyr1.tyBtnRgt.bRtCompl = TRUE THEN
				tyP0930MagConv1.tyNavi2Lyr1.tyBtnLeft.bRtCompl				:= FALSE;
				tyP0930MagConv1.tyNavi2Lyr1.tyBtnLeft.bValue				:= FALSE;
				tyP0930MagConv1.tyNavi2Lyr1.tyBtnRgt.bRtCompl				:= FALSE;
				tyP0930MagConv1.tyNavi2Lyr1.tyBtnRgt.bValue					:= FALSE;
				eChgPage													:= UIP0931MagConv2;
				bDispMagConv1	:= FALSE;
				bDispMagConv2	:= TRUE;
				bDispMagConv3	:= FALSE;

			END_IF

		ULMagTriple:
			IF tyP0930MagConv1.tyNavi3Lyr1.tyBtnBack.bRtCompl = TRUE THEN
				tyP0930MagConv1.tyNavi3Lyr1.tyBtnBack.bRtCompl	:= FALSE;
				tyP0930MagConv1.tyNavi3Lyr1.tyBtnBack.bValue		:= FALSE;

				eChgPage	:= UIP0920MtrNPneuCtrl;
				bDispMagConv1	:= TRUE;
				bDispMagConv2	:= FALSE;
				bDispMagConv3	:= FALSE;

			ELSIF tyP0930MagConv1.tyNavi3Lyr1.tyBtnLeft.bRtCompl = TRUE THEN
				tyP0930MagConv1.tyNavi3Lyr1.tyBtnLeft.bRtCompl				:= FALSE;
				tyP0930MagConv1.tyNavi3Lyr1.tyBtnLeft.bValue				:= FALSE;
				eChgPage													:= UIP0932MagConv3;
				bDispMagConv1	:= FALSE;
				bDispMagConv2	:= FALSE;
				bDispMagConv3	:= TRUE;

			ELSIF tyP0930MagConv1.tyNavi3Lyr1.tyBtnRgt.bRtCompl = TRUE THEN
				tyP0930MagConv1.tyNavi3Lyr1.tyBtnRgt.bRtCompl				:= FALSE;
				tyP0930MagConv1.tyNavi3Lyr1.tyBtnRgt.bValue					:= FALSE;
				eChgPage													:= UIP0931MagConv2;
				bDispMagConv1	:= FALSE;
				bDispMagConv2	:= TRUE;
				bDispMagConv3	:= FALSE;

			END_IF

		END_CASE

END_ACTION
```

#### Act_OptP0930MagConv1ChgLyr.st
```iecst
ACTION Act_OptP0930MagConv1ChgLyr:

	IF p_tyNtParamCurr.bMagAutoVerifyPrep THEN
		IF tyP0930MagConv1.tyCom.tyBtnSwitch.bRtCompl THEN
			tyP0930MagConv1.tyCom.tyBtnSwitch.bRtCompl	:= FALSE;

			IF tyP0930MagConv1.tyCom.tyBtnSwitch.bValue = TRUE THEN
				fUIInRtStatOff(ADR(tyP0930MagConv1.tyDC.tyLyr.uiRtStat));
				fUIInRtStatHide(ADR(tyP0930MagConv1.tyFB.tyLyr.uiRtStat));
			ELSE
				fUIInRtStatHide(ADR(tyP0930MagConv1.tyDC.tyLyr.uiRtStat));
				fUIInRtStatOff(ADR(tyP0930MagConv1.tyFB.tyLyr.uiRtStat));
			END_IF

		END_IF
	ELSE
		IF tyP0930MagConv1.tyCom.tyBtnSwitch.bRtCompl THEN
			tyP0930MagConv1.tyCom.tyBtnSwitch.bRtCompl	:= FALSE;

			IF tyP0930MagConv1.tyCom.tyBtnSwitch.bValue = TRUE THEN
				fUIInRtStatOff(ADR(tyP0930MagConv1.tyDC.tyLyrWithoutSelClamp.uiRtStat));
				fUIInRtStatHide(ADR(tyP0930MagConv1.tyFB.tyLyrWithoutSelClamp.uiRtStat));
			ELSE
				fUIInRtStatHide(ADR(tyP0930MagConv1.tyDC.tyLyrWithoutSelClamp.uiRtStat));
				fUIInRtStatOff(ADR(tyP0930MagConv1.tyFB.tyLyrWithoutSelClamp.uiRtStat));
			END_IF

		END_IF
	END_IF

END_ACTION
```

#### Act_OptP0930MagConv1Sen.st
```iecst
ACTION Act_OptP0930MagConv1Sen:
	// connect sensors to inputs
	tyP0930MagConv1.tyCom.tyBtnMagPresentSen.bValue			:= p_tyDI.bMagPresentSen1;
	tyP0930MagConv1.tyCom.tyBtnMagConvEntSen.bValue			:= p_tyDI.bMagConvEntSen1;
	tyP0930MagConv1.tyCom.tyBtnMagAIVPosSen1.bValue			:= p_tyDI.bMag1AIVInPosSen1;
	tyP0930MagConv1.tyCom.tyBtnMagAIVPosSen2.bValue			:= p_tyDI.bMag1AIVInPosSen2;
	tyP0930MagConv1.tyCom.tyBtnMagOrientationChkSen1.bValue	:= p_tyDI.bMag1OrientChkSen1;
	tyP0930MagConv1.tyCom.tyBtnMagOrientationChkSen2.bValue	:= p_tyDI.bMag1OrientChkSen2;

	tyP0930MagConv1.tyCom.tyBtnFixedClampRS.bValue			:= p_tyDI.bMag1FixedClampRS;
	tyP0930MagConv1.tyCom.tyBtnFixedUnclampRS.bValue		:= p_tyDI.bMag1FixedUnclampRS;
	tyP0930MagConv1.tyCom.tyBtnRemoteClampRS.bValue			:= p_tyDI.bMag1RemoteClampRS;
	tyP0930MagConv1.tyCom.tyBtnRemoteUnclampRS.bValue		:= p_tyDI.bMag1RemoteUnclampRS;

	tyP0930MagConv1.tyCom.tyBtnSelUnclampRS.bValue			:= p_tyDI.bMag1SelUnClampRS;

	tyP0930MagConv1.tyCom.tyBtnCAB717Sen.bValue				:= p_tyDI.bMagConvCAB717MagSen1;
	tyP0930MagConv1.tyCom.tyBtnMagSmallSen.bValue			:= p_tyDI.bMagConvSmallMagSen1;
	tyP0930MagConv1.tyCom.tyBtnMagLargeSen.bValue			:= p_tyDI.bMagConvLargeMagSen1;

	tyP0930MagConv1.tyCom.tyBtnMagDetectSen.bValue			:= p_tyDI.bMag1FixedClampSen;
//	tyP0930MagConv1.tyCom.tyBtnMagDetectSen.uiRtStat.0		:= NOT p_tyNtParamCurr.bProjFixClprMagDetectSenPrep;

	//MagHeightCheckSensor
	IF p_tyNtParamCurr.bMagAutoVerifyPrep = TRUE THEN
		tyP0930MagConv1.tyCom.tyBtnHeightSen.bValue			:= p_tyDI.bMagConvHeightSen1;
	ELSE
		tyP0930MagConv1.tyCom.tyBtnHeightSen.bValue			:= p_tyDI.bHighMagDetSen1;
	END_IF;

	//Machine Bitmap
	IF p_tyNtParamCurr.eProjMag = ULMagDual AND p_tyNtParamCurr.bMagAutoVerifyPrep = FALSE THEN
		IF tyP0930MagConv1.tyFB.tyBtnFixedClamp.bRtCompl
			OR tyP0930MagConv1.tyDC.tyBtnFixedClamp.bRtCompl THEN

			tyP0930MagConv1.tyCom.tyBitmapMc.uiValueIdx	:= 107;

		ELSIF tyP0930MagConv1.tyFB.tyBtnFixedUnclamp.bRtCompl
			OR tyP0930MagConv1.tyDC.tyBtnFixedUnclamp.bRtCompl THEN

			tyP0930MagConv1.tyCom.tyBitmapMc.uiValueIdx	:= 106;

		ELSIF tyP0930MagConv1.tyFB.tyBtnRemoteClamp.bRtCompl
			OR tyP0930MagConv1.tyDC.tyBtnRemoteClamp.bRtCompl THEN

			tyP0930MagConv1.tyCom.tyBitmapMc.uiValueIdx	:= 112;

		ELSIF tyP0930MagConv1.tyFB.tyBtnRemoteUnclamp.bRtCompl
			OR tyP0930MagConv1.tyDC.tyBtnRemoteUnclamp.bRtCompl THEN

			tyP0930MagConv1.tyCom.tyBitmapMc.uiValueIdx	:= 111;

		ELSIF tyP0930MagConv1.tyFB.tyBtnEnt.bRtCompl OR tyP0930MagConv1.tyFB.tyBtnExit.bRtCompl OR tyP0930MagConv1.tyFB.tyBtnStop.bRtCompl
			OR tyP0930MagConv1.tyDC.tyBtnMagIn.bRtCompl OR tyP0930MagConv1.tyDC.tyBtnMagOut.bRtCompl OR tyP0930MagConv1.tyDC.tyBtnStop.bRtCompl THEN

			tyP0930MagConv1.tyCom.tyBitmapMc.uiValueIdx	:= 105;

		END_IF

	ELSIF p_tyNtParamCurr.bMagAutoVerifyPrep AND p_tyNtParamCurr.bProjMagAWPrep = FALSE THEN
		IF tyP0930MagConv1.tyFB.tyBtnFixedClamp.bRtCompl
			OR tyP0930MagConv1.tyDC.tyBtnFixedClamp.bRtCompl THEN

			tyP0930MagConv1.tyCom.tyBitmapMc.uiValueIdx	:= 22;

		ELSIF tyP0930MagConv1.tyFB.tyBtnFixedUnclamp.bRtCompl
			OR tyP0930MagConv1.tyDC.tyBtnFixedUnclamp.bRtCompl THEN

			tyP0930MagConv1.tyCom.tyBitmapMc.uiValueIdx	:= 23;

		ELSIF tyP0930MagConv1.tyFB.tyBtnRemoteClamp.bRtCompl
			 OR tyP0930MagConv1.tyDC.tyBtnRemoteClamp.bRtCompl THEN

			tyP0930MagConv1.tyCom.tyBitmapMc.uiValueIdx	:= 17;

		ELSIF tyP0930MagConv1.tyFB.tyBtnRemoteUnclamp.bRtCompl
			OR tyP0930MagConv1.tyDC.tyBtnRemoteUnclamp.bRtCompl THEN

			tyP0930MagConv1.tyCom.tyBitmapMc.uiValueIdx	:= 16;

		ELSIF tyP0930MagConv1.tyFB.tyBtnSelClamp.bRtCompl
			OR tyP0930MagConv1.tyDC.tyBtnSelClamp.bRtCompl THEN

			tyP0930MagConv1.tyCom.tyBitmapMc.uiValueIdx	:= 29;

		ELSIF tyP0930MagConv1.tyFB.tyBtnSelUnclamp.bRtCompl
			OR tyP0930MagConv1.tyDC.tyBtnSelUnclamp.bRtCompl THEN

			tyP0930MagConv1.tyCom.tyBitmapMc.uiValueIdx	:= 28;

		ELSIF tyP0930MagConv1.tyFB.tyBtnEnt.bRtCompl OR tyP0930MagConv1.tyFB.tyBtnExit.bRtCompl OR tyP0930MagConv1.tyFB.tyBtnStop.bRtCompl
			OR tyP0930MagConv1.tyDC.tyBtnMagIn.bRtCompl OR tyP0930MagConv1.tyDC.tyBtnMagOut.bRtCompl OR tyP0930MagConv1.tyDC.tyBtnStop.bRtCompl THEN

			tyP0930MagConv1.tyCom.tyBitmapMc.uiValueIdx	:= 0;

		END_IF

	ELSIF p_tyNtParamCurr.eProjMag = ULMagTriple AND  p_tyNtParamCurr.bMagAutoVerifyPrep AND p_tyNtParamCurr.bProjMagAWPrep AND p_tyNtParamCurr.bProjMotorizedPusherPrep = FALSE THEN
		IF tyP0930MagConv1.tyFB.tyBtnFixedClamp.bRtCompl
				OR tyP0930MagConv1.tyDC.tyBtnFixedClamp.bRtCompl THEN

				tyP0930MagConv1.tyCom.tyBitmapMc.uiValueIdx	:= 46;

			ELSIF tyP0930MagConv1.tyFB.tyBtnFixedUnclamp.bRtCompl
				OR tyP0930MagConv1.tyDC.tyBtnFixedUnclamp.bRtCompl THEN

				tyP0930MagConv1.tyCom.tyBitmapMc.uiValueIdx	:= 47;

			ELSIF tyP0930MagConv1.tyFB.tyBtnRemoteClamp.bRtCompl
				OR tyP0930MagConv1.tyDC.tyBtnRemoteClamp.bRtCompl THEN

				tyP0930MagConv1.tyCom.tyBitmapMc.uiValueIdx	:= 59;

			ELSIF tyP0930MagConv1.tyFB.tyBtnRemoteUnclamp.bRtCompl
				OR tyP0930MagConv1.tyDC.tyBtnRemoteUnclamp.bRtCompl THEN

				tyP0930MagConv1.tyCom.tyBitmapMc.uiValueIdx	:= 58;

			ELSIF tyP0930MagConv1.tyFB.tyBtnSelClamp.bRtCompl
				OR tyP0930MagConv1.tyDC.tyBtnSelClamp.bRtCompl THEN

				tyP0930MagConv1.tyCom.tyBitmapMc.uiValueIdx	:= 41;

			ELSIF tyP0930MagConv1.tyFB.tyBtnSelUnclamp.bRtCompl
				OR tyP0930MagConv1.tyDC.tyBtnSelUnclamp.bRtCompl THEN

				tyP0930MagConv1.tyCom.tyBitmapMc.uiValueIdx	:= 40;

			ELSIF tyP0930MagConv1.tyFB.tyBtnEnt.bRtCompl OR tyP0930MagConv1.tyFB.tyBtnExit.bRtCompl OR tyP0930MagConv1.tyFB.tyBtnStop.bRtCompl
				OR tyP0930MagConv1.tyDC.tyBtnMagIn.bRtCompl OR tyP0930MagConv1.tyDC.tyBtnMagOut.bRtCompl OR tyP0930MagConv1.tyDC.tyBtnStop.bRtCompl THEN

				tyP0930MagConv1.tyCom.tyBitmapMc.uiValueIdx	:= 3;

			END_IF

		ELSIF p_tyNtParamCurr.eProjMag = ULMagTriple AND p_tyNtParamCurr.bMagAutoVerifyPrep =FALSE  AND p_tyNtParamCurr.bProjMagAWPrep = FALSE AND p_tyNtParamCurr.bProjMotorizedPusherPrep THEN
			IF tyP0930MagConv1.tyFB.tyBtnFixedClamp.bRtCompl
					OR tyP0930MagConv1.tyDC.tyBtnFixedClamp.bRtCompl THEN

					IF p_tyNtParamCurr.bCurtainSenPrep THEN
						tyP0930MagConv1.tyCom.tyBitmapMc.uiValueIdx	:= 232;
					ELSE
						tyP0930MagConv1.tyCom.tyBitmapMc.uiValueIdx	:= 203;
				    END_IF

				ELSIF tyP0930MagConv1.tyFB.tyBtnFixedUnclamp.bRtCompl
					OR tyP0930MagConv1.tyDC.tyBtnFixedUnclamp.bRtCompl THEN

					IF p_tyNtParamCurr.bCurtainSenPrep THEN
						tyP0930MagConv1.tyCom.tyBitmapMc.uiValueIdx	:= 232;
					ELSE
						tyP0930MagConv1.tyCom.tyBitmapMc.uiValueIdx	:= 202;
					END_IF

				ELSIF tyP0930MagConv1.tyFB.tyBtnRemoteClamp.bRtCompl
					OR tyP0930MagConv1.tyDC.tyBtnRemoteClamp.bRtCompl THEN

					IF p_tyNtParamCurr.bCurtainSenPrep THEN
						tyP0930MagConv1.tyCom.tyBitmapMc.uiValueIdx	:= 232;
					ELSE
						tyP0930MagConv1.tyCom.tyBitmapMc.uiValueIdx	:= 217;
					END_IF

				ELSIF tyP0930MagConv1.tyFB.tyBtnRemoteUnclamp.bRtCompl
					OR tyP0930MagConv1.tyDC.tyBtnRemoteUnclamp.bRtCompl THEN

					IF p_tyNtParamCurr.bCurtainSenPrep THEN
						tyP0930MagConv1.tyCom.tyBitmapMc.uiValueIdx	:= 232;
					ELSE
						tyP0930MagConv1.tyCom.tyBitmapMc.uiValueIdx	:= 216;
					END_IF

//				ELSIF tyP0930MagConv1.tyFB.tyBtnSelClamp.bRtCompl
//					OR tyP0930MagConv1.tyDC.tyBtnSelClamp.bRtCompl THEN
//
//					tyP0930MagConv1.tyCom.tyBitmapMc.uiValueIdx	:= 41;
//
//				ELSIF tyP0930MagConv1.tyFB.tyBtnSelUnclamp.bRtCompl
//					OR tyP0930MagConv1.tyDC.tyBtnSelUnclamp.bRtCompl THEN
//
//					tyP0930MagConv1.tyCom.tyBitmapMc.uiValueIdx	:= 40;
//
				ELSIF tyP0930MagConv1.tyFB.tyBtnEnt.bRtCompl OR tyP0930MagConv1.tyFB.tyBtnExit.bRtCompl OR tyP0930MagConv1.tyFB.tyBtnStop.bRtCompl
					OR tyP0930MagConv1.tyDC.tyBtnMagIn.bRtCompl OR tyP0930MagConv1.tyDC.tyBtnMagOut.bRtCompl OR tyP0930MagConv1.tyDC.tyBtnStop.bRtCompl THEN

					IF p_tyNtParamCurr.bCurtainSenPrep THEN
						tyP0930MagConv1.tyCom.tyBitmapMc.uiValueIdx	:= 233;
					ELSE
						tyP0930MagConv1.tyCom.tyBitmapMc.uiValueIdx	:= 203;
					END_IF

				END_IF

		ELSIF p_tyNtParamCurr.eProjMag = ULMagDual AND p_tyNtParamCurr.bMagAutoVerifyPrep THEN
			IF tyP0930MagConv1.tyFB.tyBtnFixedClamp.bRtCompl
				OR tyP0930MagConv1.tyDC.tyBtnFixedClamp.bRtCompl THEN

				tyP0930MagConv1.tyCom.tyBitmapMc.uiValueIdx	:= 146;

			ELSIF tyP0930MagConv1.tyFB.tyBtnFixedUnclamp.bRtCompl
				OR tyP0930MagConv1.tyDC.tyBtnFixedUnclamp.bRtCompl THEN

				tyP0930MagConv1.tyCom.tyBitmapMc.uiValueIdx	:= 147;

			ELSIF tyP0930MagConv1.tyFB.tyBtnRemoteClamp.bRtCompl
				OR tyP0930MagConv1.tyDC.tyBtnRemoteClamp.bRtCompl THEN

				tyP0930MagConv1.tyCom.tyBitmapMc.uiValueIdx	:= 159;

			ELSIF tyP0930MagConv1.tyFB.tyBtnRemoteUnclamp.bRtCompl
				OR tyP0930MagConv1.tyDC.tyBtnRemoteUnclamp.bRtCompl THEN

				tyP0930MagConv1.tyCom.tyBitmapMc.uiValueIdx	:= 158;

			ELSIF tyP0930MagConv1.tyFB.tyBtnSelClamp.bRtCompl
				OR tyP0930MagConv1.tyDC.tyBtnSelClamp.bRtCompl THEN

				tyP0930MagConv1.tyCom.tyBitmapMc.uiValueIdx	:= 141;

			ELSIF tyP0930MagConv1.tyFB.tyBtnSelUnclamp.bRtCompl
				OR tyP0930MagConv1.tyDC.tyBtnSelUnclamp.bRtCompl THEN

				tyP0930MagConv1.tyCom.tyBitmapMc.uiValueIdx	:= 140;

			ELSIF tyP0930MagConv1.tyFB.tyBtnEnt.bRtCompl OR tyP0930MagConv1.tyFB.tyBtnExit.bRtCompl OR tyP0930MagConv1.tyFB.tyBtnStop.bRtCompl
				OR tyP0930MagConv1.tyDC.tyBtnMagIn.bRtCompl OR tyP0930MagConv1.tyDC.tyBtnMagOut.bRtCompl OR tyP0930MagConv1.tyDC.tyBtnStop.bRtCompl THEN

				tyP0930MagConv1.tyCom.tyBitmapMc.uiValueIdx	:= 103;

			END_IF
		END_IF

//	IF p_tyNtParamCurr.eProjMag = ULMagTriple AND p_tyNtParamCurr.bMagAutoVerifyPrep = FALSE THEN
//		IF tyP0930MagConv1.tyCom.tyBitmapMc.uiValueIdx < 100 THEN
//			tyP0930MagConv1.tyCom.tyBitmapMc.uiValueIdx	:= tyP0930MagConv1.tyCom.tyBitmapMc.uiValueIdx + 100;
//		END_IF
//	ELSIF p_tyNtParamCurr.eProjMag = ULMagTriple AND p_tyNtParamCurr.bMagAutoVerifyPrep = TRUE THEN
//			IF tyP0930MagConv1.tyCom.tyBitmapMc.uiValueIdx < 200 THEN
//				tyP0930MagConv1.tyCom.tyBitmapMc.uiValueIdx	:= tyP0930MagConv1.tyCom.tyBitmapMc.uiValueIdx + 200;
//			END_IF
//	END_IF

END_ACTION
```

#### Act_OptP0930MagConv1FB.st
```iecst
ACTION Act_OptP0930MagConv1FB:

	//Magazine Conveyor
	IF tyP0930MagConv1.tyFB.tyBtnStop.bRtCompl = TRUE THEN
		eMagConv2Clp1Act	:= MagConv2ClpActStop;

		IF p_eMagConv2Clp1Stat = MagConv2ClpActStop AND p_eMagConv2Clp1Status = Done THEN
			eMagConv2Clp1Act	:= MagConv2ClpActIdle;

			tyP0930MagConv1.tyFB.tyBtnEnt.bRtCompl	:= FALSE;
			tyP0930MagConv1.tyFB.tyBtnEnt.bValue	:= FALSE;
			tyP0930MagConv1.tyFB.tyBtnEnt.bRtLk		:= FALSE;

			tyP0930MagConv1.tyFB.tyBtnExit.bRtCompl	:= FALSE;
			tyP0930MagConv1.tyFB.tyBtnExit.bValue	:= FALSE;
			tyP0930MagConv1.tyFB.tyBtnExit.bRtLk	:= FALSE;

			tyP0930MagConv1.tyFB.tyBtnStop.bRtCompl	:= FALSE;
			tyP0930MagConv1.tyFB.tyBtnStop.bValue	:= TRUE;
			tyP0930MagConv1.tyFB.tyBtnStop.bRtLk	:= TRUE;
		END_IF

	ELSIF tyP0930MagConv1.tyFB.tyBtnEnt.bRtCompl = TRUE THEN
		tyP0930MagConv1.tyFB.tyBtnEnt.bValue	:= TRUE;
		tyP0930MagConv1.tyFB.tyBtnEnt.bRtLk		:= TRUE;

		tyP0930MagConv1.tyFB.tyBtnStop.bValue	:= FALSE;
		tyP0930MagConv1.tyFB.tyBtnStop.bRtLk	:= FALSE;

		eMagConv2Clp1Act	:= MagConv2ClpActEnt;

		IF p_eMagConv2Clp1Stat = MagConv2ClpActEnt AND p_eMagConv2Clp1Status = Done THEN
			eMagConv2Clp1Act	:= MagConv2ClpActIdle;

			tyP0930MagConv1.tyFB.tyBtnEnt.bRtCompl	:= FALSE;

			tyP0930MagConv1.tyFB.tyBtnEnt.bValue	:= FALSE;
			tyP0930MagConv1.tyFB.tyBtnEnt.bRtLk		:= FALSE;

			tyP0930MagConv1.tyFB.tyBtnStop.bValue	:= TRUE;
			tyP0930MagConv1.tyFB.tyBtnStop.bRtLk	:= TRUE;
		END_IF

	ELSIF (p_eMagConv2Clp1Stat = MagConv2ClpActPreExit AND p_eMagConv2Clp1Status = Done) THEN
		eMagConv2Clp1Act	:= MagConv2ClpActIdle;

			tyP0930MagConv1.tyFB.tyBtnExit.bRtCompl	:= FALSE;

			tyP0930MagConv1.tyFB.tyBtnExit.bValue	:= FALSE;
			tyP0930MagConv1.tyFB.tyBtnExit.bRtLk	:= FALSE;

			tyP0930MagConv1.tyFB.tyBtnStop.bValue	:= TRUE;
			tyP0930MagConv1.tyFB.tyBtnStop.bRtLk	:= TRUE;

	ELSIF (p_eMagConv2Clp1Stat = MagConv2ClpActExit AND p_eMagConv2Clp1Status = Done) THEN
			eMagConv2Clp1Act	:= MagConv2ClpActIdle;

			tyP0930MagConv1.tyFB.tyBtnExit.bRtCompl	:= FALSE;

			tyP0930MagConv1.tyFB.tyBtnExit.bValue	:= FALSE;
			tyP0930MagConv1.tyFB.tyBtnExit.bRtLk	:= FALSE;

			tyP0930MagConv1.tyFB.tyBtnStop.bValue	:= TRUE;
			tyP0930MagConv1.tyFB.tyBtnStop.bRtLk	:= TRUE;

	ELSIF tyP0930MagConv1.tyFB.tyBtnExit.bRtCompl = TRUE THEN
		tyP0930MagConv1.tyFB.tyBtnExit.bRtCompl	:= FALSE;
		tyP0930MagConv1.tyFB.tyBtnExit.bValue	:= TRUE;
		tyP0930MagConv1.tyFB.tyBtnExit.bRtLk	:= TRUE;

		tyP0930MagConv1.tyFB.tyBtnStop.bValue	:= FALSE;
		tyP0930MagConv1.tyFB.tyBtnStop.bRtLk	:= FALSE;

		IF p_tyDI.bMagConvEntSen1  THEN
			eMagConv2Clp1Act	:= MagConv2ClpActExit;
		ELSE
			IF p_tyDI.bMagPresentSen1 THEN
				eMagConv2Clp1Act	:= MagConv2ClpActPreExit;
			ELSE
				eMagConv2Clp1Act	:= MagConv2ClpActExit;
			END_IF
		END_IF
	END_IF

	//Magazine Clamper
	IF tyP0930MagConv1.tyCom.tyBtnSwitch.bValue = FALSE THEN

		//Fixed
		IF tyP0930MagConv1.tyFB.tyBtnFixedUnclamp.bRtCompl = TRUE THEN
			tyP0930MagConv1.tyFB.tyBtnFixedUnclamp.bRtCompl	:= FALSE;

			tyP0930MagConv1.tyFB.tyBtnFixedUnclamp.bValue	:= TRUE;
			tyP0930MagConv1.tyFB.tyBtnFixedClamp.bValue		:= FALSE;

		ELSIF tyP0930MagConv1.tyFB.tyBtnFixedClamp.bRtCompl = TRUE THEN
			tyP0930MagConv1.tyFB.tyBtnFixedClamp.bRtCompl	:= FALSE;

			tyP0930MagConv1.tyFB.tyBtnFixedClamp.bValue		:= TRUE;
			tyP0930MagConv1.tyFB.tyBtnFixedUnclamp.bValue	:= FALSE;

		END_IF

		//Remote
		IF tyP0930MagConv1.tyFB.tyBtnRemoteUnclamp.bRtCompl = TRUE THEN
			tyP0930MagConv1.tyFB.tyBtnRemoteUnclamp.bRtCompl	:= FALSE;

			tyP0930MagConv1.tyFB.tyBtnRemoteUnclamp.bValue	:= TRUE;
			tyP0930MagConv1.tyFB.tyBtnRemoteClamp.bValue	:= FALSE;

		ELSIF tyP0930MagConv1.tyFB.tyBtnRemoteClamp.bRtCompl = TRUE THEN
			tyP0930MagConv1.tyFB.tyBtnRemoteClamp.bRtCompl	:= FALSE;

			tyP0930MagConv1.tyFB.tyBtnRemoteClamp.bValue	:= TRUE;
			tyP0930MagConv1.tyFB.tyBtnRemoteUnclamp.bValue	:= FALSE;

		END_IF

		//Sel
		IF tyP0930MagConv1.tyFB.tyBtnSelUnclamp.bRtCompl = TRUE THEN
			tyP0930MagConv1.tyFB.tyBtnSelUnclamp.bRtCompl	:= FALSE;

			tyP0930MagConv1.tyFB.tyBtnSelUnclamp.bValue	:= TRUE;
			tyP0930MagConv1.tyFB.tyBtnSelClamp.bValue	:= FALSE;

		ELSIF tyP0930MagConv1.tyFB.tyBtnSelClamp.bRtCompl = TRUE THEN
			tyP0930MagConv1.tyFB.tyBtnSelClamp.bRtCompl	:= FALSE;

			tyP0930MagConv1.tyFB.tyBtnSelClamp.bValue	:= TRUE;
			tyP0930MagConv1.tyFB.tyBtnSelUnclamp.bValue	:= FALSE;

		END_IF

		// Fixed Clamper
		IF tyP0930MagConv1.tyFB.tyBtnFixedUnclamp.bValue = TRUE THEN

			eMagConv2Clp1Act	:= MagConv2ClpActFixClprUnclamp;

			IF p_eMagConv2Clp1Stat = MagConv2ClpActFixClprUnclamp AND p_eMagConv2Clp1Status = Done THEN

				eMagConv2Clp1Act	:= MagConv2ClpActIdle;

				tyP0930MagConv1.tyFB.tyBtnFixedUnclamp.bValue	:= FALSE;

			ELSIF p_eMagConv2Clp1Status = Error THEN

				tyP0930MagConv1.tyFB.tyBtnFixedUnclamp.bValue	:= FALSE;

			END_IF

		ELSIF tyP0930MagConv1.tyFB.tyBtnFixedClamp.bValue = TRUE THEN
			eMagConv2Clp1Act	:= MagConv2ClpActFixClprClamp;

			IF p_eMagConv2Clp1Stat = MagConv2ClpActFixClprClamp AND p_eMagConv2Clp1Status = Done THEN

				eMagConv2Clp1Act	:= MagConv2ClpActIdle;

				tyP0930MagConv1.tyFB.tyBtnFixedClamp.bValue := FALSE;

			ELSIF p_eMagConv2Clp1Status = Error THEN
				tyP0930MagConv1.tyFB.tyBtnFixedClamp.bValue := FALSE;

			END_IF

		END_IF

		//Remote Clamper
		IF tyP0930MagConv1.tyFB.tyBtnRemoteUnclamp.bValue = TRUE THEN

			eMagConv2Clp1Act	:= MagConv2ClpActRmtClprUnclamp;

			IF p_eMagConv2Clp1Stat = MagConv2ClpActRmtClprUnclamp AND p_eMagConv2Clp1Status = Done THEN

				eMagConv2Clp1Act	:= MagConv2ClpActIdle;

				tyP0930MagConv1.tyFB.tyBtnRemoteUnclamp.bValue	:= FALSE;

			ELSIF p_eMagConv2Clp1Status = Error THEN

				tyP0930MagConv1.tyFB.tyBtnRemoteUnclamp.bValue	:= FALSE;

			END_IF

		ELSIF tyP0930MagConv1.tyFB.tyBtnRemoteClamp.bValue = TRUE THEN
			eMagConv2Clp1Act	:= MagConv2ClpActRmtClprClamp;

			IF p_eMagConv2Clp1Stat = MagConv2ClpActRmtClprClamp AND p_eMagConv2Clp1Status = Done THEN

				eMagConv2Clp1Act	:= MagConv2ClpActIdle;

				tyP0930MagConv1.tyFB.tyBtnRemoteClamp.bValue := FALSE;

			ELSIF p_eMagConv2Clp1Status = Error THEN
				tyP0930MagConv1.tyFB.tyBtnRemoteClamp.bValue := FALSE;

			END_IF

		END_IF

		//Sel Clamper
		IF tyP0930MagConv1.tyFB.tyBtnSelUnclamp.bValue = TRUE THEN

			eMagConvSelClp1Act	:= PneuActExt;

			IF p_eSelClamp1Stat = PneuActExt AND p_eSelClamp1Status = Done THEN

				eMagConvSelClp1Act	:= PneuActIdle;

				tyP0930MagConv1.tyFB.tyBtnSelUnclamp.bValue	:= FALSE;

			ELSIF p_eSelClamp1Status = Error THEN

				tyP0930MagConv1.tyFB.tyBtnSelUnclamp.bValue	:= FALSE;

			END_IF

		ELSIF tyP0930MagConv1.tyFB.tyBtnSelClamp.bValue = TRUE THEN
			eMagConvSelClp1Act	:= PneuActRet;

			IF p_eSelClamp1Stat = PneuActRet AND p_eSelClamp1Status = Done THEN

				eMagConvSelClp1Act	:= PneuActIdle;

				tyP0930MagConv1.tyFB.tyBtnSelClamp.bValue	:= FALSE;

			ELSIF p_eSelClamp1Status = Error THEN
				tyP0930MagConv1.tyFB.tyBtnSelClamp.bValue	:= FALSE;

			END_IF

		END_IF

		//Update Status
		tyP0930MagConv1.tyDC.tyBtnFixedUnclamp.bValue	:= NOT p_bMagConv2Clp1ClprFixClampCtrl;
		tyP0930MagConv1.tyDC.tyBtnFixedClamp.bValue		:= p_bMagConv2Clp1ClprFixClampCtrl;
		tyP0930MagConv1.tyDC.tyBtnRemoteUnclamp.bValue	:= NOT p_bMagConv2Clp1ClprRmtClampCtrl;
		tyP0930MagConv1.tyDC.tyBtnRemoteClamp.bValue	:= p_bMagConv2Clp1ClprRmtClampCtrl;

		tyP0930MagConv1.tyDC.tyBtnSelUnclamp.bRtCompl	:= FALSE;
		tyP0930MagConv1.tyDC.tyBtnSelClamp.bRtCompl		:= FALSE;
		tyP0930MagConv1.tyDC.tyBtnSelUnclamp.bValue	:= p_bSelClamp1RetCtrl;
		tyP0930MagConv1.tyDC.tyBtnSelClamp.bValue	:= p_bSelClamp1ExtCtrl;
	END_IF

	//Mask
	IF p_tyUsrMgmtCurrAccessRgt.bManualFBOnly THEN

		fUIInRtStatOff(ADR(tyP0930MagConv1.tyCom.tyBtnSwitch.uiMaskRtStat));

	ELSE

	IF p_eMagConv2Clp1Status = Error THEN

		fUIInRtStatOff(ADR(tyP0930MagConv1.tyFB.tyBtnEnt.uiMaskRtStat));
		fUIInRtStatOff(ADR(tyP0930MagConv1.tyFB.tyBtnExit.uiMaskRtStat));
		fUIInRtStatOff(ADR(tyP0930MagConv1.tyFB.tyBtnFixedClamp.uiMaskRtStat));
		fUIInRtStatOff(ADR(tyP0930MagConv1.tyFB.tyBtnFixedUnclamp.uiMaskRtStat));
		fUIInRtStatOff(ADR(tyP0930MagConv1.tyFB.tyBtnRemoteClamp.uiMaskRtStat));
		fUIInRtStatOff(ADR(tyP0930MagConv1.tyFB.tyBtnRemoteUnclamp.uiMaskRtStat));
		fUIInRtStatOff(ADR(tyP0930MagConv1.tyFB.tyBtnSelClamp.uiMaskRtStat));
		fUIInRtStatOff(ADR(tyP0930MagConv1.tyFB.tyBtnSelUnclamp.uiMaskRtStat));
		fUIInRtStatHide(ADR(tyP0930MagConv1.tyCom.tyBtnSwitch.uiMaskRtStat));

	ELSIF tyP0930MagConv1.tyFB.tyBtnEnt.bRtCompl = TRUE THEN

		fUIInRtStatHide(ADR(tyP0930MagConv1.tyFB.tyBtnEnt.uiMaskRtStat));
		fUIInRtStatOff(ADR(tyP0930MagConv1.tyFB.tyBtnExit.uiMaskRtStat));
		fUIInRtStatOff(ADR(tyP0930MagConv1.tyFB.tyBtnFixedClamp.uiMaskRtStat));
		fUIInRtStatOff(ADR(tyP0930MagConv1.tyFB.tyBtnFixedUnclamp.uiMaskRtStat));
		fUIInRtStatOff(ADR(tyP0930MagConv1.tyFB.tyBtnRemoteClamp.uiMaskRtStat));
		fUIInRtStatOff(ADR(tyP0930MagConv1.tyFB.tyBtnRemoteUnclamp.uiMaskRtStat));
		fUIInRtStatOff(ADR(tyP0930MagConv1.tyFB.tyBtnSelClamp.uiMaskRtStat));
		fUIInRtStatOff(ADR(tyP0930MagConv1.tyFB.tyBtnSelUnclamp.uiMaskRtStat));
		fUIInRtStatOff(ADR(tyP0930MagConv1.tyCom.tyBtnSwitch.uiMaskRtStat));

	ELSIF tyP0930MagConv1.tyFB.tyBtnExit.bRtCompl = TRUE THEN

		fUIInRtStatOff(ADR(tyP0930MagConv1.tyFB.tyBtnEnt.uiMaskRtStat));
		fUIInRtStatHide(ADR(tyP0930MagConv1.tyFB.tyBtnExit.uiMaskRtStat));
		fUIInRtStatOff(ADR(tyP0930MagConv1.tyFB.tyBtnFixedClamp.uiMaskRtStat));
		fUIInRtStatOff(ADR(tyP0930MagConv1.tyFB.tyBtnFixedUnclamp.uiMaskRtStat));
		fUIInRtStatOff(ADR(tyP0930MagConv1.tyFB.tyBtnRemoteClamp.uiMaskRtStat));
		fUIInRtStatOff(ADR(tyP0930MagConv1.tyFB.tyBtnRemoteUnclamp.uiMaskRtStat));
		fUIInRtStatOff(ADR(tyP0930MagConv1.tyFB.tyBtnSelClamp.uiMaskRtStat));
		fUIInRtStatOff(ADR(tyP0930MagConv1.tyFB.tyBtnSelUnclamp.uiMaskRtStat));
		fUIInRtStatOff(ADR(tyP0930MagConv1.tyCom.tyBtnSwitch.uiMaskRtStat));

	ELSIF tyP0930MagConv1.tyFB.tyBtnFixedClamp.bValue = TRUE OR tyP0930MagConv1.tyFB.tyBtnRemoteClamp.bValue = TRUE
			OR tyP0930MagConv1.tyFB.tyBtnFixedUnclamp.bValue = TRUE OR tyP0930MagConv1.tyFB.tyBtnRemoteUnclamp.bValue = TRUE
			OR tyP0930MagConv1.tyFB.tyBtnSelUnclamp.bValue = TRUE OR tyP0930MagConv1.tyFB.tyBtnSelClamp.bValue = TRUE
			THEN

		fUIInRtStatOff(ADR(tyP0930MagConv1.tyFB.tyBtnEnt.uiMaskRtStat));
		fUIInRtStatOff(ADR(tyP0930MagConv1.tyFB.tyBtnExit.uiMaskRtStat));
		fUIInRtStatHide(ADR(tyP0930MagConv1.tyFB.tyBtnFixedClamp.uiMaskRtStat));
		fUIInRtStatHide(ADR(tyP0930MagConv1.tyFB.tyBtnFixedUnclamp.uiMaskRtStat));
		fUIInRtStatHide(ADR(tyP0930MagConv1.tyFB.tyBtnRemoteClamp.uiMaskRtStat));
		fUIInRtStatHide(ADR(tyP0930MagConv1.tyFB.tyBtnRemoteUnclamp.uiMaskRtStat));
		fUIInRtStatHide(ADR(tyP0930MagConv1.tyFB.tyBtnSelClamp.uiMaskRtStat));
		fUIInRtStatHide(ADR(tyP0930MagConv1.tyFB.tyBtnSelUnclamp.uiMaskRtStat));
		fUIInRtStatOff(ADR(tyP0930MagConv1.tyCom.tyBtnSwitch.uiMaskRtStat));

	ELSE

		fUIInRtStatHide(ADR(tyP0930MagConv1.tyFB.tyBtnEnt.uiMaskRtStat));
		fUIInRtStatHide(ADR(tyP0930MagConv1.tyFB.tyBtnExit.uiMaskRtStat));
		fUIInRtStatHide(ADR(tyP0930MagConv1.tyFB.tyBtnFixedClamp.uiMaskRtStat));
		fUIInRtStatHide(ADR(tyP0930MagConv1.tyFB.tyBtnFixedUnclamp.uiMaskRtStat));
		fUIInRtStatHide(ADR(tyP0930MagConv1.tyFB.tyBtnRemoteClamp.uiMaskRtStat));
		fUIInRtStatHide(ADR(tyP0930MagConv1.tyFB.tyBtnRemoteUnclamp.uiMaskRtStat));
		fUIInRtStatHide(ADR(tyP0930MagConv1.tyFB.tyBtnSelClamp.uiMaskRtStat));
		fUIInRtStatHide(ADR(tyP0930MagConv1.tyFB.tyBtnSelUnclamp.uiMaskRtStat));
		fUIInRtStatHide(ADR(tyP0930MagConv1.tyCom.tyBtnSwitch.uiMaskRtStat));

	END_IF
END_IF

	IF p_tyDI.bMagConvCAB717MagSen1 THEN
			fUIInRtStatOff(ADR(tyP0930MagConv1.tyFB.tyBtnSelClamp.uiMaskRtStat));
	END_IF

	IF p_bMagConv2Clp1ClprFixClampCtrl OR p_bMagConv2Clp1ClprRmtClampCtrl THEN
		fUIInRtStatOff(ADR(tyP0930MagConv1.tyFB.tyBtnEnt.uiMaskRtStat));
		fUIInRtStatOff(ADR(tyP0930MagConv1.tyFB.tyBtnExit.uiMaskRtStat));
	END_IF

END_ACTION
```

#### Act_OptP0930MagConv1FBStat.st
```iecst
ACTION Act_OptP0930MagConv1FBStat:

IF tyP0930MagConv1.tyFB.tyBtnFixedClamp.bValue = TRUE OR tyP0930MagConv1.tyFB.tyBtnRemoteClamp.bValue = TRUE
	OR tyP0930MagConv1.tyFB.tyBtnFixedUnclamp.bValue = TRUE OR tyP0930MagConv1.tyFB.tyBtnRemoteUnclamp.bValue = TRUE
		THEN
		tyP0930MagConv1.tyFB.tyStringStat.sValue	:= p_sMagConv2Clp1StatTxt;
ELSIF (tyP0930MagConv1.tyFB.tyBtnFixedClamp.bValue = FALSE AND  tyP0930MagConv1.tyFB.tyBtnRemoteClamp.bValue = FALSE
		AND tyP0930MagConv1.tyFB.tyBtnFixedUnclamp.bValue = FALSE AND  tyP0930MagConv1.tyFB.tyBtnRemoteUnclamp.bValue = FALSE
		AND p_eMagConv2Clp1Status <> Busy)
		THEN
		tyP0930MagConv1.tyFB.tyStringStat.sValue	:= p_sMagConv2Clp1StatTxt;
ELSIF tyP0930MagConv1.tyFB.tyBtnSelUnclamp.bValue = TRUE OR tyP0930MagConv1.tyFB.tyBtnSelClamp.bValue = TRUE
		THEN
		tyP0930MagConv1.tyFB.tyStringStat.sValue	:= p_sSelClamp1StatTxt;
END_IF

END_ACTION
```

#### Act_OptP0930MagConv1DC.st
```iecst
ACTION Act_OptP0930MagConv1DC:

	//Magazine Conveyor
	IF tyP0930MagConv1.tyDC.tyBtnStop.bRtCompl = TRUE THEN
		eMagConv2Clp1Act	:= MagConv2ClpActStop;

		IF p_eMagConv2Clp1Stat = MagConv2ClpActStop AND p_eMagConv2Clp1Status = Done THEN
			eMagConv2Clp1Act	:= MagConv2ClpActIdle;

			tyP0930MagConv1.tyDC.tyBtnStop.bRtCompl		:= FALSE;
			tyP0930MagConv1.tyDC.tyBtnStop.bValue		:= TRUE;
			tyP0930MagConv1.tyDC.tyBtnStop.bRtLk		:= TRUE;

			tyP0930MagConv1.tyDC.tyBtnMagIn.bRtCompl	:= FALSE;
			tyP0930MagConv1.tyDC.tyBtnMagIn.bValue		:= FALSE;
			tyP0930MagConv1.tyDC.tyBtnMagIn.bRtLk		:= FALSE;

			tyP0930MagConv1.tyDC.tyBtnMagOut.bRtCompl	:= FALSE;
			tyP0930MagConv1.tyDC.tyBtnMagOut.bValue		:= FALSE;
			tyP0930MagConv1.tyDC.tyBtnMagOut.bRtLk		:= FALSE;
		END_IF

	ELSIF tyP0930MagConv1.tyDC.tyBtnMagIn.bRtCompl = TRUE THEN
		tyP0930MagConv1.tyDC.tyBtnMagIn.bValue	:= TRUE;
		tyP0930MagConv1.tyDC.tyBtnMagIn.bRtLk	:= TRUE;

		tyP0930MagConv1.tyDC.tyBtnStop.bValue	:= FALSE;
		tyP0930MagConv1.tyDC.tyBtnStop.bRtLk	:= FALSE;

		IF p_tyNtParamCurr.eProjMagConvDir = ConvDirLToR OR p_tyNtParamCurr.eProjMagConvDir = ConvDirLToL THEN

			eMagConv2Clp1Act	:= MagConv2ClpActSetMtrSigOnOrLToR;

			IF p_eMagConv2Clp1Stat = MagConv2ClpActSetMtrSigOnOrLToR AND p_eMagConv2Clp1Status = Done THEN
				eMagConv2Clp1Act	:= MagConv2ClpActIdle;

				tyP0930MagConv1.tyDC.tyBtnMagIn.bRtCompl	:= FALSE;
			END_IF

		ELSE

			eMagConv2Clp1Act	:= MagConv2ClpActSetMtrDirOrRToL;

			IF p_eMagConv2Clp1Stat = MagConv2ClpActSetMtrDirOrRToL AND p_eMagConv2Clp1Status = Done THEN
				eMagConv2Clp1Act	:= MagConv2ClpActIdle;

				tyP0930MagConv1.tyDC.tyBtnMagIn.bRtCompl	:= FALSE;
			END_IF

		END_IF

	ELSIF tyP0930MagConv1.tyDC.tyBtnMagOut.bRtCompl = TRUE THEN
		tyP0930MagConv1.tyDC.tyBtnMagOut.bValue	:= TRUE;
		tyP0930MagConv1.tyDC.tyBtnMagOut.bRtLk	:= TRUE;

		tyP0930MagConv1.tyDC.tyBtnStop.bValue	:= FALSE;
		tyP0930MagConv1.tyDC.tyBtnStop.bRtLk	:= FALSE;

		IF p_tyNtParamCurr.eProjMagConvDir = ConvDirLToR OR p_tyNtParamCurr.eProjMagConvDir = ConvDirRToR THEN

			eMagConv2Clp1Act	:= MagConv2ClpActSetMtrSigOnOrLToR;

			IF p_eMagConv2Clp1Stat = MagConv2ClpActSetMtrSigOnOrLToR AND p_eMagConv2Clp1Status = Done THEN
				eMagConv2Clp1Act	:= MagConv2ClpActIdle;

				tyP0930MagConv1.tyDC.tyBtnMagOut.bRtCompl	:= FALSE;
			END_IF

		ELSE

			eMagConv2Clp1Act	:= MagConv2ClpActSetMtrDirOrRToL;

			IF p_eMagConv2Clp1Stat = MagConv2ClpActSetMtrDirOrRToL AND p_eMagConv2Clp1Status = Done THEN
				eMagConv2Clp1Act	:= MagConv2ClpActIdle;

				tyP0930MagConv1.tyDC.tyBtnMagOut.bRtCompl	:= FALSE;
			END_IF

		END_IF

	END_IF

	//Magazine Clamper
	IF tyP0930MagConv1.tyCom.tyBtnSwitch.bValue = TRUE THEN
		IF p_bSelClamp1TwoCtrlOut = FALSE THEN
			IF tyP0930MagConv1.tyDC.tyBtnSelUnclamp.bRtCompl = TRUE THEN
				tyP0930MagConv1.tyDC.tyBtnSelUnclamp.bValue := TRUE;
				tyP0930MagConv1.tyDC.tyBtnSelClamp.bValue := FALSE;

				eMagConvSelClp1Act	:= PneuActSetExt;

				IF p_eSelClamp1Stat = PneuActSetExt AND p_eSelClamp1Status = Done THEN
					eMagConvSelClp1Act	:= PneuActIdle;

					tyP0930MagConv1.tyDC.tyBtnSelUnclamp.bRtCompl	:= FALSE;
				END_IF

			ELSIF tyP0930MagConv1.tyDC.tyBtnSelClamp.bRtCompl = TRUE THEN
				tyP0930MagConv1.tyDC.tyBtnSelClamp.bValue := TRUE;
				tyP0930MagConv1.tyDC.tyBtnSelUnclamp.bValue := FALSE;

				eMagConvSelClp1Act	:= PneuActSetRet;

				IF p_eSelClamp1Stat = PneuActSetRet AND p_eSelClamp1Status = Done THEN
					eMagConvSelClp1Act	:= PneuActIdle;

					tyP0930MagConv1.tyDC.tyBtnSelClamp.bRtCompl	:= FALSE;
				END_IF
			END_IF

		ELSE
			IF (tyP0930MagConv1.tyDC.tyBtnSelUnclamp.bRtCompl = TRUE) OR (tyP0930MagConv1.tyDC.tyBtnSelClamp.bRtCompl = TRUE) THEN
				IF (tyP0930MagConv1.tyDC.tyBtnSelUnclamp.bValue = TRUE) AND (tyP0930MagConv1.tyDC.tyBtnSelClamp.bValue = TRUE) THEN
					eMagConvSelClp1Act	:= PneuActSetAll;

					IF p_eSelClamp1Stat = PneuActSetAll AND p_eSelClamp1Status = Done THEN
						eMagConvSelClp1Act	:= PneuActIdle;

						tyP0930MagConv1.tyDC.tyBtnSelUnclamp.bRtCompl		:= FALSE;
						tyP0930MagConv1.tyDC.tyBtnSelClamp.bRtCompl			:= FALSE;
					END_IF
		/////////i edited the ret to ext
				ELSIF (tyP0930MagConv1.tyDC.tyBtnSelUnclamp.bValue = TRUE) AND (tyP0930MagConv1.tyDC.tyBtnSelClamp.bValue = FALSE) THEN
					eMagConvSelClp1Act	:= PneuActSetExt;(**)

					IF p_eSelClamp1Stat = PneuActSetExt (**) AND p_eSelClamp1Status = Done THEN
						eMagConvSelClp1Act	:= PneuActIdle;

						tyP0930MagConv1.tyDC.tyBtnSelUnclamp.bRtCompl		:= FALSE;
						tyP0930MagConv1.tyDC.tyBtnSelClamp.bRtCompl			:= FALSE;
					END_IF

				ELSIF (tyP0930MagConv1.tyDC.tyBtnSelUnclamp.bValue = FALSE) AND (tyP0930MagConv1.tyDC.tyBtnSelClamp.bValue = TRUE) THEN
						eMagConvSelClp1Act	:= PneuActSetRet;

					IF p_eSelClamp1Stat = PneuActSetRet AND p_eSelClamp1Status = Done THEN
						eMagConvSelClp1Act	:= PneuActIdle;

						tyP0930MagConv1.tyDC.tyBtnSelUnclamp.bRtCompl		:= FALSE;
						tyP0930MagConv1.tyDC.tyBtnSelClamp.bRtCompl			:= FALSE;
					END_IF
					///////
				ELSE
					eMagConvSelClp1Act	:= PneuActRstAll;

					IF p_eSelClamp1Stat = PneuActRstAll AND p_eSelClamp1Status = Done THEN
						eMagConvSelClp1Act	:= PneuActIdle;

						tyP0930MagConv1.tyDC.tyBtnSelUnclamp.bRtCompl		:= FALSE;
						tyP0930MagConv1.tyDC.tyBtnSelClamp.bRtCompl			:= FALSE;
					END_IF

				END_IF
			END_IF
		END_IF

		IF p_bMagConv2Clp1ClprTwoOutputCtrl = FALSE THEN

			//Fixed
			IF tyP0930MagConv1.tyDC.tyBtnFixedClamp.bRtCompl = TRUE THEN
				tyP0930MagConv1.tyDC.tyBtnFixedClamp.bValue		:= TRUE;
				tyP0930MagConv1.tyDC.tyBtnFixedUnclamp.bValue	:= FALSE;

				eMagConv2Clp1Act	:= MagConv2ClpActFixClprSetClamp;

				IF p_eMagConv2Clp1Stat = MagConv2ClpActFixClprSetClamp AND p_eMagConv2Clp1Status = Done THEN
					eMagConv2Clp1Act	:= MagConv2ClpActIdle;

					tyP0930MagConv1.tyDC.tyBtnFixedClamp.bRtCompl	:= FALSE;
				END_IF

			ELSIF tyP0930MagConv1.tyDC.tyBtnFixedUnclamp.bRtCompl = TRUE THEN
				tyP0930MagConv1.tyDC.tyBtnFixedUnclamp.bValue	:= TRUE;
				tyP0930MagConv1.tyDC.tyBtnFixedClamp.bValue		:= FALSE;

				eMagConv2Clp1Act	:= MagConv2ClpActFixClprSetUnclamp;

				IF p_eMagConv2Clp1Stat = MagConv2ClpActFixClprSetUnclamp AND p_eMagConv2Clp1Status = Done THEN
					eMagConv2Clp1Act	:= MagConv2ClpActIdle;

					tyP0930MagConv1.tyDC.tyBtnFixedUnclamp.bRtCompl	:= FALSE;
				END_IF

			END_IF

			//Remote
			IF tyP0930MagConv1.tyDC.tyBtnRemoteClamp.bRtCompl = TRUE THEN
				tyP0930MagConv1.tyDC.tyBtnRemoteClamp.bValue		:= TRUE;
				tyP0930MagConv1.tyDC.tyBtnRemoteUnclamp.bValue		:= FALSE;

				eMagConv2Clp1Act	:= MagConv2ClpActRmtClprSetClamp;

				IF p_eMagConv2Clp1Stat = MagConv2ClpActRmtClprSetClamp AND p_eMagConv2Clp1Status = Done THEN
					eMagConv2Clp1Act	:= MagConv2ClpActIdle;

					tyP0930MagConv1.tyDC.tyBtnRemoteClamp.bRtCompl	:= FALSE;
				END_IF

			ELSIF tyP0930MagConv1.tyDC.tyBtnRemoteUnclamp.bRtCompl = TRUE THEN
				tyP0930MagConv1.tyDC.tyBtnRemoteUnclamp.bValue	:= TRUE;
				tyP0930MagConv1.tyDC.tyBtnRemoteClamp.bValue	:= FALSE;

				eMagConv2Clp1Act	:= MagConv2ClpActRmtClprSetUnclamp;

				IF p_eMagConv2Clp1Stat = MagConv2ClpActRmtClprSetUnclamp AND p_eMagConv2Clp1Status = Done THEN
					eMagConv2Clp1Act	:= MagConv2ClpActIdle;

					tyP0930MagConv1.tyDC.tyBtnRemoteUnclamp.bRtCompl	:= FALSE;
				END_IF

			END_IF

		ELSE

			//Fixed
			IF (tyP0930MagConv1.tyDC.tyBtnFixedClamp.bRtCompl = TRUE) OR (tyP0930MagConv1.tyDC.tyBtnFixedUnclamp.bRtCompl = TRUE) THEN

				IF (tyP0930MagConv1.tyDC.tyBtnFixedClamp.bValue = TRUE) AND (tyP0930MagConv1.tyDC.tyBtnFixedUnclamp.bValue = TRUE) THEN

					eMagConv2Clp1Act	:= MagConv2ClpActFixClprSetAll;

					IF p_eMagConv2Clp1Stat = MagConv2ClpActFixClprSetAll AND p_eMagConv2Clp1Status = Done THEN

						eMagConv2Clp1Act	:= MagConv2ClpActIdle;

						tyP0930MagConv1.tyDC.tyBtnFixedClamp.bRtCompl	:= FALSE;
						tyP0930MagConv1.tyDC.tyBtnFixedUnclamp.bRtCompl	:= FALSE;
					END_IF

				ELSIF (tyP0930MagConv1.tyDC.tyBtnFixedClamp.bValue = TRUE) AND (tyP0930MagConv1.tyDC.tyBtnFixedUnclamp.bValue = FALSE) THEN
					eMagConv2Clp1Act	:= MagConv2ClpActFixClprSetClamp;

					IF p_eMagConv2Clp1Stat = MagConv2ClpActFixClprSetClamp AND p_eMagConv2Clp1Status = Done THEN

						eMagConv2Clp1Act	:= MagConv2ClpActIdle;

						tyP0930MagConv1.tyDC.tyBtnFixedClamp.bRtCompl	:= FALSE;
						tyP0930MagConv1.tyDC.tyBtnFixedUnclamp.bRtCompl	:= FALSE;
					END_IF

				ELSIF (tyP0930MagConv1.tyDC.tyBtnFixedClamp.bValue = FALSE) AND (tyP0930MagConv1.tyDC.tyBtnFixedUnclamp.bValue = TRUE) THEN
					eMagConv2Clp1Act	:= MagConv2ClpActFixClprSetUnclamp;

					IF p_eMagConv2Clp1Stat = MagConv2ClpActFixClprSetUnclamp AND p_eMagConv2Clp1Status = Done THEN

						eMagConv2Clp1Act	:= MagConv2ClpActIdle;

						tyP0930MagConv1.tyDC.tyBtnFixedClamp.bRtCompl	:= FALSE;
						tyP0930MagConv1.tyDC.tyBtnFixedUnclamp.bRtCompl	:= FALSE;
					END_IF

				ELSE
					eMagConv2Clp1Act	:= MagConv2ClpActFixClprRstAll;

					IF p_eMagConv2Clp1Stat = MagConv2ClpActFixClprRstAll AND p_eMagConv2Clp1Status = Done THEN

						eMagConv2Clp1Act	:= MagConv2ClpActIdle;

						tyP0930MagConv1.tyDC.tyBtnFixedClamp.bRtCompl	:= FALSE;
						tyP0930MagConv1.tyDC.tyBtnFixedUnclamp.bRtCompl	:= FALSE;
					END_IF

				END_IF

				//Remote
				IF (tyP0930MagConv1.tyDC.tyBtnRemoteClamp.bRtCompl = TRUE) OR (tyP0930MagConv1.tyDC.tyBtnRemoteUnclamp.bRtCompl = TRUE) THEN

					IF (tyP0930MagConv1.tyDC.tyBtnRemoteClamp.bValue = TRUE) AND (tyP0930MagConv1.tyDC.tyBtnRemoteUnclamp.bValue = TRUE) THEN

						eMagConv2Clp1Act	:= MagConv2ClpActRmtClprSetAll;

						IF p_eMagConv2Clp1Stat = MagConv2ClpActRmtClprSetAll AND p_eMagConv2Clp1Status = Done THEN

							eMagConv2Clp1Act	:= MagConv2ClpActIdle;

							tyP0930MagConv1.tyDC.tyBtnRemoteClamp.bRtCompl		:= FALSE;
							tyP0930MagConv1.tyDC.tyBtnRemoteUnclamp.bRtCompl	:= FALSE;
						END_IF

					ELSIF (tyP0930MagConv1.tyDC.tyBtnRemoteClamp.bValue = TRUE) AND (tyP0930MagConv1.tyDC.tyBtnRemoteUnclamp.bValue = FALSE) THEN
						eMagConv2Clp1Act	:= MagConv2ClpActRmtClprSetClamp;

						IF p_eMagConv2Clp1Stat = MagConv2ClpActRmtClprSetClamp AND p_eMagConv2Clp1Status = Done THEN

							eMagConv2Clp1Act	:= MagConv2ClpActIdle;

							tyP0930MagConv1.tyDC.tyBtnRemoteClamp.bRtCompl	:= FALSE;
							tyP0930MagConv1.tyDC.tyBtnRemoteUnclamp.bRtCompl	:= FALSE;
						END_IF

					ELSIF (tyP0930MagConv1.tyDC.tyBtnRemoteClamp.bValue = FALSE) AND (tyP0930MagConv1.tyDC.tyBtnRemoteUnclamp.bValue = TRUE) THEN
						eMagConv2Clp1Act	:= MagConv2ClpActRmtClprSetUnclamp;

						IF p_eMagConv2Clp1Stat = MagConv2ClpActRmtClprSetUnclamp AND p_eMagConv2Clp1Status = Done THEN

							eMagConv2Clp1Act	:= MagConv2ClpActIdle;

							tyP0930MagConv1.tyDC.tyBtnRemoteClamp.bRtCompl	:= FALSE;
							tyP0930MagConv1.tyDC.tyBtnRemoteUnclamp.bRtCompl	:= FALSE;
						END_IF

					ELSE
						eMagConv2Clp1Act	:= MagConv2ClpActRmtClprRstAll;

						IF p_eMagConv2Clp1Stat = MagConv2ClpActRmtClprRstAll AND p_eMagConv2Clp1Status = Done THEN

							eMagConv2Clp1Act	:= MagConv2ClpActIdle;

							tyP0930MagConv1.tyDC.tyBtnRemoteClamp.bRtCompl	:= FALSE;
							tyP0930MagConv1.tyDC.tyBtnRemoteUnclamp.bRtCompl	:= FALSE;
						END_IF

					END_IF
				END_IF

			END_IF

		END_IF

		//Fixed
		tyP0930MagConv1.tyFB.tyBtnFixedClamp.bRtCompl		:= FALSE;
		tyP0930MagConv1.tyFB.tyBtnFixedClamp.bValue			:= FALSE;
		tyP0930MagConv1.tyFB.tyBtnFixedUnclamp.bRtCompl		:= FALSE;
		tyP0930MagConv1.tyFB.tyBtnFixedUnclamp.bValue		:= FALSE;

		//Remote
		tyP0930MagConv1.tyFB.tyBtnRemoteClamp.bRtCompl		:= FALSE;
		tyP0930MagConv1.tyFB.tyBtnRemoteClamp.bValue		:= FALSE;
		tyP0930MagConv1.tyFB.tyBtnRemoteUnclamp.bRtCompl	:= FALSE;
		tyP0930MagConv1.tyFB.tyBtnRemoteUnclamp.bValue		:= FALSE;

		//Top
		tyP0930MagConv1.tyFB.tyBtnSelClamp.bRtCompl		:= FALSE;
		tyP0930MagConv1.tyFB.tyBtnSelClamp.bValue		:= FALSE;
		tyP0930MagConv1.tyFB.tyBtnSelUnclamp.bRtCompl	:= FALSE;
		tyP0930MagConv1.tyFB.tyBtnSelUnclamp.bValue		:= FALSE;
	END_IF

	//Mask
	IF p_eMagConv2Clp1Status = Error THEN

		fUIInRtStatOff(ADR(tyP0930MagConv1.tyDC.tyBtnMagIn.uiMaskRtStat));
		fUIInRtStatOff(ADR(tyP0930MagConv1.tyDC.tyBtnMagOut.uiMaskRtStat));
		fUIInRtStatOff(ADR(tyP0930MagConv1.tyDC.tyBtnFixedClamp.uiMaskRtStat));
		fUIInRtStatOff(ADR(tyP0930MagConv1.tyDC.tyBtnFixedUnclamp.uiMaskRtStat));
		fUIInRtStatOff(ADR(tyP0930MagConv1.tyDC.tyBtnRemoteClamp.uiMaskRtStat));
		fUIInRtStatOff(ADR(tyP0930MagConv1.tyDC.tyBtnRemoteUnclamp.uiMaskRtStat));
		fUIInRtStatOff(ADR(tyP0930MagConv1.tyDC.tyBtnSelClamp.uiMaskRtStat));
		fUIInRtStatOff(ADR(tyP0930MagConv1.tyDC.tyBtnSelUnclamp.uiMaskRtStat));

	ELSIF tyP0930MagConv1.tyDC.tyBtnMagIn.bValue = TRUE THEN

		fUIInRtStatHide(ADR(tyP0930MagConv1.tyDC.tyBtnMagIn.uiMaskRtStat));
		fUIInRtStatOff(ADR(tyP0930MagConv1.tyDC.tyBtnMagOut.uiMaskRtStat));
		fUIInRtStatOff(ADR(tyP0930MagConv1.tyDC.tyBtnFixedClamp.uiMaskRtStat));
		fUIInRtStatOff(ADR(tyP0930MagConv1.tyDC.tyBtnFixedUnclamp.uiMaskRtStat));
		fUIInRtStatOff(ADR(tyP0930MagConv1.tyDC.tyBtnRemoteClamp.uiMaskRtStat));
		fUIInRtStatOff(ADR(tyP0930MagConv1.tyDC.tyBtnRemoteUnclamp.uiMaskRtStat));
		fUIInRtStatOff(ADR(tyP0930MagConv1.tyDC.tyBtnSelClamp.uiMaskRtStat));
		fUIInRtStatOff(ADR(tyP0930MagConv1.tyDC.tyBtnSelUnclamp.uiMaskRtStat));

	ELSIF tyP0930MagConv1.tyDC.tyBtnMagOut.bValue = TRUE THEN

		fUIInRtStatOff(ADR(tyP0930MagConv1.tyDC.tyBtnMagIn.uiMaskRtStat));
		fUIInRtStatHide(ADR(tyP0930MagConv1.tyDC.tyBtnMagOut.uiMaskRtStat));
		fUIInRtStatOff(ADR(tyP0930MagConv1.tyDC.tyBtnFixedClamp.uiMaskRtStat));
		fUIInRtStatOff(ADR(tyP0930MagConv1.tyDC.tyBtnFixedUnclamp.uiMaskRtStat));
		fUIInRtStatOff(ADR(tyP0930MagConv1.tyDC.tyBtnRemoteClamp.uiMaskRtStat));
		fUIInRtStatOff(ADR(tyP0930MagConv1.tyDC.tyBtnRemoteUnclamp.uiMaskRtStat));
		fUIInRtStatOff(ADR(tyP0930MagConv1.tyDC.tyBtnSelClamp.uiMaskRtStat));
		fUIInRtStatOff(ADR(tyP0930MagConv1.tyDC.tyBtnSelUnclamp.uiMaskRtStat));

	ELSE

		fUIInRtStatHide(ADR(tyP0930MagConv1.tyDC.tyBtnMagIn.uiMaskRtStat));
		fUIInRtStatHide(ADR(tyP0930MagConv1.tyDC.tyBtnMagOut.uiMaskRtStat));
		fUIInRtStatHide(ADR(tyP0930MagConv1.tyDC.tyBtnFixedClamp.uiMaskRtStat));
		fUIInRtStatHide(ADR(tyP0930MagConv1.tyDC.tyBtnFixedUnclamp.uiMaskRtStat));
		fUIInRtStatHide(ADR(tyP0930MagConv1.tyDC.tyBtnRemoteClamp.uiMaskRtStat));
		fUIInRtStatHide(ADR(tyP0930MagConv1.tyDC.tyBtnRemoteUnclamp.uiMaskRtStat));
		fUIInRtStatHide(ADR(tyP0930MagConv1.tyDC.tyBtnSelClamp.uiMaskRtStat));
		fUIInRtStatHide(ADR(tyP0930MagConv1.tyDC.tyBtnSelUnclamp.uiMaskRtStat));

	END_IF

END_ACTION
```

#### Act_OptP0930RstMnl.st
```iecst
ACTION Act_OptP0930RstMnl:

	IF EDGEPOS((bManualMod = FALSE) OR (p_eMagConv2Clp1Status = Error)) THEN

		eMagConv2Clp1Act	:= MagConv2ClpActIdle;
		eMagConvSelClp1Act	:= PneuActIdle;
		//Magazine Conveyor
		//FB
		tyP0930MagConv1.tyFB.tyBtnEnt.bRtCompl				:= FALSE;
		tyP0930MagConv1.tyFB.tyBtnExit.bRtCompl				:= FALSE;
		tyP0930MagConv1.tyFB.tyBtnStop.bRtCompl				:= FALSE;

		tyP0930MagConv1.tyFB.tyBtnEnt.bValue				:= FALSE;
		tyP0930MagConv1.tyFB.tyBtnExit.bValue				:= FALSE;
		tyP0930MagConv1.tyFB.tyBtnStop.bValue				:= TRUE;

		tyP0930MagConv1.tyFB.tyBtnEnt.bRtLk					:= FALSE;
		tyP0930MagConv1.tyFB.tyBtnExit.bRtLk				:= FALSE;
		tyP0930MagConv1.tyFB.tyBtnStop.bRtLk				:= TRUE;

		tyP0930MagConv1.tyFB.tyBtnEnt.uiMaskRtStat.0		:= TRUE;
		tyP0930MagConv1.tyFB.tyBtnExit.uiMaskRtStat.0		:= TRUE;
		tyP0930MagConv1.tyCom.tyBtnSwitch.uiMaskRtStat.0	:= TRUE;

		//Direct
		tyP0930MagConv1.tyDC.tyBtnMagIn.bRtCompl			:= FALSE;
		tyP0930MagConv1.tyDC.tyBtnMagOut.bRtCompl			:= FALSE;
		tyP0930MagConv1.tyDC.tyBtnStop.bRtCompl				:= FALSE;

		tyP0930MagConv1.tyDC.tyBtnMagIn.bValue				:= FALSE;
		tyP0930MagConv1.tyDC.tyBtnMagOut.bValue				:= FALSE;
		tyP0930MagConv1.tyDC.tyBtnStop.bValue				:= TRUE;

		tyP0930MagConv1.tyDC.tyBtnMagIn.bRtLk				:= FALSE;
		tyP0930MagConv1.tyDC.tyBtnMagOut.bRtLk				:= FALSE;
		tyP0930MagConv1.tyDC.tyBtnStop.bRtLk				:= TRUE;

		tyP0930MagConv1.tyDC.tyBtnMagIn.uiMaskRtStat.0		:= TRUE;
		tyP0930MagConv1.tyDC.tyBtnMagOut.uiMaskRtStat.0		:= TRUE;
		tyP0930MagConv1.tyCom.tyBtnSwitch.uiMaskRtStat.0	:= TRUE;

		//Magazine Clamper
		//FB
		//Top
		tyP0930MagConv1.tyFB.tyBtnFixedClamp.bRtCompl			:= FALSE;
		tyP0930MagConv1.tyFB.tyBtnFixedUnclamp.bRtCompl			:= FALSE;

		tyP0930MagConv1.tyFB.tyBtnFixedClamp.bValue				:= FALSE;
		tyP0930MagConv1.tyFB.tyBtnFixedUnclamp.bValue			:= FALSE;

		//Remote
		tyP0930MagConv1.tyFB.tyBtnRemoteClamp.bRtCompl			:= FALSE;
		tyP0930MagConv1.tyFB.tyBtnRemoteUnclamp.bRtCompl		:= FALSE;

		tyP0930MagConv1.tyFB.tyBtnRemoteClamp.bValue			:= FALSE;
		tyP0930MagConv1.tyFB.tyBtnRemoteUnclamp.bValue			:= FALSE;

		//Top
		tyP0930MagConv1.tyFB.tyBtnSelClamp.bRtCompl			:= FALSE;
		tyP0930MagConv1.tyFB.tyBtnSelUnclamp.bRtCompl		:= FALSE;

		tyP0930MagConv1.tyFB.tyBtnSelClamp.bValue			:= FALSE;
		tyP0930MagConv1.tyFB.tyBtnSelUnclamp.bValue			:= FALSE;

		tyP0930MagConv1.tyFB.tyBtnFixedClamp.uiMaskRtStat.0		:= TRUE;
		tyP0930MagConv1.tyFB.tyBtnFixedUnclamp.uiMaskRtStat.0	:= TRUE;
		tyP0930MagConv1.tyFB.tyBtnRemoteClamp.uiMaskRtStat.0	:= TRUE;
		tyP0930MagConv1.tyFB.tyBtnRemoteUnclamp.uiMaskRtStat.0	:= TRUE;
		tyP0930MagConv1.tyFB.tyBtnSelClamp.uiMaskRtStat.0		:= TRUE;
		tyP0930MagConv1.tyFB.tyBtnSelUnclamp.uiMaskRtStat.0		:= TRUE;

		tyP0930MagConv1.tyCom.tyBtnSwitch.uiMaskRtStat.0		:= TRUE;

		//Direct
		//Fixed
		tyP0930MagConv1.tyDC.tyBtnFixedClamp.bRtCompl			:= FALSE;
		tyP0930MagConv1.tyDC.tyBtnFixedUnclamp.bRtCompl			:= FALSE;

		tyP0930MagConv1.tyDC.tyBtnFixedClamp.bValue				:= FALSE;
		tyP0930MagConv1.tyDC.tyBtnFixedUnclamp.bValue			:= FALSE;

		//Remote
		tyP0930MagConv1.tyDC.tyBtnRemoteClamp.bRtCompl			:= FALSE;
		tyP0930MagConv1.tyDC.tyBtnRemoteUnclamp.bRtCompl		:= FALSE;

		tyP0930MagConv1.tyDC.tyBtnRemoteClamp.bValue			:= FALSE;
		tyP0930MagConv1.tyDC.tyBtnRemoteUnclamp.bValue			:= FALSE;

		//Top
		tyP0930MagConv1.tyDC.tyBtnSelClamp.bRtCompl				:= FALSE;
		tyP0930MagConv1.tyDC.tyBtnSelUnclamp.bRtCompl			:= FALSE;

		tyP0930MagConv1.tyDC.tyBtnSelClamp.bValue				:= FALSE;
		tyP0930MagConv1.tyDC.tyBtnSelUnclamp.bValue				:= FALSE;

		tyP0930MagConv1.tyDC.tyBtnFixedClamp.uiMaskRtStat.0		:= TRUE;
		tyP0930MagConv1.tyDC.tyBtnFixedUnclamp.uiMaskRtStat.0	:= TRUE;
		tyP0930MagConv1.tyDC.tyBtnRemoteClamp.uiMaskRtStat.0	:= TRUE;
		tyP0930MagConv1.tyDC.tyBtnRemoteUnclamp.uiMaskRtStat.0	:= TRUE;
		tyP0930MagConv1.tyDC.tyBtnSelClamp.uiMaskRtStat.0		:= TRUE;
		tyP0930MagConv1.tyDC.tyBtnSelUnclamp.uiMaskRtStat.0		:= TRUE;

		tyP0930MagConv1.tyCom.tyBtnSwitch.uiMaskRtStat.0		:= TRUE;

	END_IF

	IF EDGEPOS(bManualMod = FALSE) THEN
		tyP0930MagConv1.tyCom.tyBtnSwitch.bValue := FALSE;

		IF p_tyNtParamCurr.bMagAutoVerifyPrep = FALSE THEN
			fUIInRtStatHide(ADR(tyP0930MagConv1.tyDC.tyLyrWithoutSelClamp.uiRtStat));
			fUIInRtStatOff(ADR(tyP0930MagConv1.tyFB.tyLyrWithoutSelClamp.uiRtStat));
		ELSE

			fUIInRtStatHide(ADR(tyP0930MagConv1.tyDC.tyLyr.uiRtStat));
			fUIInRtStatOff(ADR(tyP0930MagConv1.tyFB.tyLyr.uiRtStat));
		END_IF
	END_IF

END_ACTION
```

#### Act_EntP0931Disp.st
```iecst
ACTION Act_EntP0931Disp:

	//Access Address
	p_tyC0002FullMask ACCESS ADR(tyP0931MagConv2.tyFullMaskHide);

	//p_tyC0004Navi ACCESS ADR(tyP0931MagConv2.tyNaviBack);

	CASE p_tyNtParamCurr.eProjMag OF
		ULMagDual:
			p_tyC0004Navi ACCESS ADR(tyP0931MagConv2.tyNavi2Lyr2);
		ULMagTriple:
			p_tyC0004Navi ACCESS ADR(tyP0931MagConv2.tyNavi3Lyr2);
	END_CASE

	p_tyC0005Main ACCESS ADR(tyCommon.tyMain);

	p_tyC0007Notif ACCESS ADR(tyCommon.tyNotif);

	p_tyC0008MsgBox ACCESS ADR(tyP0931MagConv2.tyMsgBoxHide);

	p_tyC0009Info ACCESS ADR(tyCommon.tyInfo);

	p_tyP0931Mag2ConvCom ACCESS ADR(tyP0931MagConv2.tyCom);
	p_tyP0931Mag2ConvDC ACCESS ADR(tyP0931MagConv2.tyDC);
	p_tyP0931Mag2ConvFB ACCESS ADR(tyP0931MagConv2.tyFB);

	IF p_tyNtParamCurr.bMagAutoVerifyPrep AND p_tyNtParamCurr.bProjMagAWPrep THEN
		IF p_tyNtParamCurr.eProjMag = ULMagDual THEN
			tyP0931MagConv2.tyCom.tyBitmapMc.uiValueIdx	:= 103;
		END_IF
	ELSIF p_tyNtParamCurr.bMagAutoVerifyPrep = FALSE AND p_tyNtParamCurr.bProjMagAWPrep = FALSE THEN
		IF p_tyNtParamCurr.eProjMag = ULMagDual THEN
			tyP0931MagConv2.tyCom.tyBitmapMc.uiValueIdx	:= 107;
		END_IF
	ELSE
		tyP0931MagConv2.tyCom.tyBitmapMc.uiValueIdx	:= 234;
	END_IF

	IF p_tyNtParamCurr.bMagAutoVerifyPrep = FALSE THEN
		IF tyP0931MagConv2.tyCom.tyBtnSwitch.bValue THEN
			fUIInRtStatHide(ADR(tyP0931MagConv2.tyFB.tyLyr.uiRtStat));
			fUIInRtStatHide(ADR(tyP0931MagConv2.tyDC.tyLyr.uiRtStat));
			fUIInRtStatHide(ADR(tyP0931MagConv2.tyFB.tyLyrWithoutSelClamp.uiRtStat));
			fUIInRtStatOff(ADR(tyP0931MagConv2.tyDC.tyLyrWithoutSelClamp.uiRtStat));
		ELSE
			fUIInRtStatHide(ADR(tyP0931MagConv2.tyFB.tyLyr.uiRtStat));
			fUIInRtStatHide(ADR(tyP0931MagConv2.tyDC.tyLyr.uiRtStat));
			fUIInRtStatOff(ADR(tyP0931MagConv2.tyFB.tyLyrWithoutSelClamp.uiRtStat));
			fUIInRtStatHide(ADR(tyP0931MagConv2.tyDC.tyLyrWithoutSelClamp.uiRtStat));
		END_IF
	ELSE
		IF tyP0931MagConv2.tyCom.tyBtnSwitch.bValue THEN
			fUIInRtStatHide(ADR(tyP0931MagConv2.tyFB.tyLyr.uiRtStat));
			fUIInRtStatOff(ADR(tyP0931MagConv2.tyDC.tyLyr.uiRtStat));
			fUIInRtStatHide(ADR(tyP0931MagConv2.tyFB.tyLyrWithoutSelClamp.uiRtStat));
			fUIInRtStatHide(ADR(tyP0931MagConv2.tyDC.tyLyrWithoutSelClamp.uiRtStat));
		ELSE
			fUIInRtStatOff(ADR(tyP0931MagConv2.tyFB.tyLyr.uiRtStat));
			fUIInRtStatHide(ADR(tyP0931MagConv2.tyDC.tyLyr.uiRtStat));
			fUIInRtStatHide(ADR(tyP0931MagConv2.tyFB.tyLyrWithoutSelClamp.uiRtStat));
			fUIInRtStatHide(ADR(tyP0931MagConv2.tyDC.tyLyrWithoutSelClamp.uiRtStat));
		END_IF
	END_IF
END_ACTION
```

#### Act_OptP0931FullMask.st
```iecst
ACTION Act_OptP0931FullMask:

	IF eCurrPage = UIP0931MagConv2 THEN

		IF p_tyDI.bEStopSig = FALSE THEN
			p_tyC0002FullMask ACCESS ADR(tyP0931MagConv2.tyFullMaskEStop);

		ELSIF p_tyDI.bCoverSWSig = FALSE THEN
			p_tyC0002FullMask ACCESS ADR(tyP0931MagConv2.tyFullMaskCWSig);

		ELSIF p_tyDI.bSafetyRlySig = FALSE THEN
			p_tyC0002FullMask ACCESS ADR(tyP0931MagConv2.tyFullMaskSafetyRly);

		ELSIF p_bMag2AWEngageExtCtrl
			AND NOT p_bMagConv2Clp2ClprFixClampCtrl
			AND NOT p_bMagConv2Clp2ClprRmtClampCtrl
			THEN
			p_tyC0002FullMask ACCESS ADR(tyP0931MagConv2.tyFullMaskAWMotorEngage);

		ELSE
			p_tyC0002FullMask ACCESS ADR(tyP0931MagConv2.tyFullMaskHide);

		END_IF

	END_IF

END_ACTION
```

#### Act_OptP0931Navi.st
```iecst
ACTION Act_OptP0931Navi:

//	IF tyP0931MagConv2.tyNaviBack.tyBtnBack.bRtCompl = TRUE THEN
//		tyP0931MagConv2.tyNaviBack.tyBtnBack.bRtCompl	:= FALSE;
//		tyP0931MagConv2.tyNaviBack.tyBtnBack.bValue		:= FALSE;
//
//		eChgPage	:= UIP0920MtrNPneuCtrl;
//	END_IF

	CASE p_tyNtParamCurr.eProjMag OF
		ULMagDual:
			IF tyP0931MagConv2.tyNavi2Lyr2.tyBtnBack.bRtCompl = TRUE THEN
				tyP0931MagConv2.tyNavi2Lyr2.tyBtnBack.bRtCompl	:= FALSE;
				tyP0931MagConv2.tyNavi2Lyr2.tyBtnBack.bValue		:= FALSE;

				eChgPage	:= UIP0920MtrNPneuCtrl;
				bDispMagConv1	:= FALSE;
				bDispMagConv2	:= TRUE;
				bDispMagConv3	:= FALSE;

			ELSIF tyP0931MagConv2.tyNavi2Lyr2.tyBtnLeft.bRtCompl = TRUE OR tyP0931MagConv2.tyNavi2Lyr2.tyBtnRgt.bRtCompl = TRUE THEN
				tyP0931MagConv2.tyNavi2Lyr2.tyBtnLeft.bRtCompl				:= FALSE;
				tyP0931MagConv2.tyNavi2Lyr2.tyBtnLeft.bValue				:= FALSE;
				tyP0931MagConv2.tyNavi2Lyr2.tyBtnRgt.bRtCompl				:= FALSE;
				tyP0931MagConv2.tyNavi2Lyr2.tyBtnRgt.bValue					:= FALSE;
				eChgPage													:= UIP0930MagConv1;
				bDispMagConv1	:= TRUE;
				bDispMagConv2	:= FALSE;
				bDispMagConv3	:= FALSE;
			END_IF

		ULMagTriple:
			IF tyP0931MagConv2.tyNavi3Lyr2.tyBtnBack.bRtCompl = TRUE THEN
				tyP0931MagConv2.tyNavi3Lyr2.tyBtnBack.bRtCompl	:= FALSE;
				tyP0931MagConv2.tyNavi3Lyr2.tyBtnBack.bValue		:= FALSE;

				eChgPage	:= UIP0920MtrNPneuCtrl;
				bDispMagConv1	:= FALSE;
				bDispMagConv2	:= TRUE;
				bDispMagConv3	:= FALSE;

			ELSIF tyP0931MagConv2.tyNavi3Lyr2.tyBtnLeft.bRtCompl = TRUE THEN
				tyP0931MagConv2.tyNavi3Lyr2.tyBtnLeft.bRtCompl				:= FALSE;
				tyP0931MagConv2.tyNavi3Lyr2.tyBtnLeft.bValue				:= FALSE;
				eChgPage													:= UIP0930MagConv1;
				bDispMagConv1	:= TRUE;
				bDispMagConv2	:= FALSE;
				bDispMagConv3	:= FALSE;

			ELSIF tyP0931MagConv2.tyNavi3Lyr2.tyBtnRgt.bRtCompl = TRUE THEN
				tyP0931MagConv2.tyNavi3Lyr2.tyBtnRgt.bRtCompl				:= FALSE;
				tyP0931MagConv2.tyNavi3Lyr2.tyBtnRgt.bValue					:= FALSE;
				eChgPage													:= UIP0932MagConv3;
				bDispMagConv1	:= FALSE;
				bDispMagConv2	:= FALSE;
				bDispMagConv3	:= TRUE;
			END_IF

	END_CASE

END_ACTION
```

#### Act_OptP0931MagConv2ChgLyr.st
```iecst
ACTION Act_OptP0931MagConv2ChgLyr:

	IF p_tyNtParamCurr.bMagAutoVerifyPrep THEN
		IF tyP0931MagConv2.tyCom.tyBtnSwitch.bRtCompl THEN
			tyP0931MagConv2.tyCom.tyBtnSwitch.bRtCompl	:= FALSE;

			IF tyP0931MagConv2.tyCom.tyBtnSwitch.bValue = TRUE THEN
				fUIInRtStatOff(ADR(tyP0931MagConv2.tyDC.tyLyr.uiRtStat));
				fUIInRtStatHide(ADR(tyP0931MagConv2.tyFB.tyLyr.uiRtStat));
			ELSE
				fUIInRtStatHide(ADR(tyP0931MagConv2.tyDC.tyLyr.uiRtStat));
				fUIInRtStatOff(ADR(tyP0931MagConv2.tyFB.tyLyr.uiRtStat));
			END_IF

		END_IF
	ELSE
		IF tyP0931MagConv2.tyCom.tyBtnSwitch.bRtCompl THEN
			tyP0931MagConv2.tyCom.tyBtnSwitch.bRtCompl	:= FALSE;

			IF tyP0931MagConv2.tyCom.tyBtnSwitch.bValue = TRUE THEN
				fUIInRtStatOff(ADR(tyP0931MagConv2.tyDC.tyLyrWithoutSelClamp.uiRtStat));
				fUIInRtStatHide(ADR(tyP0931MagConv2.tyFB.tyLyrWithoutSelClamp.uiRtStat));
			ELSE
				fUIInRtStatHide(ADR(tyP0931MagConv2.tyDC.tyLyrWithoutSelClamp.uiRtStat));
				fUIInRtStatOff(ADR(tyP0931MagConv2.tyFB.tyLyrWithoutSelClamp.uiRtStat));
			END_IF

		END_IF
	END_IF

END_ACTION
```

#### Act_OptP0931MagConv2Sen.st
```iecst
ACTION Act_OptP0931MagConv2Sen:

	tyP0931MagConv2.tyCom.tyBtnMagPresentSen.bValue			:= p_tyDI.bMagPresentSen2;
	tyP0931MagConv2.tyCom.tyBtnMagConvEntSen.bValue			:= p_tyDI.bMagConvEntSen2;
	tyP0931MagConv2.tyCom.tyBtnMagAIVPosSen1.bValue			:= p_tyDI.bMag2AIVInPosSen1;
	tyP0931MagConv2.tyCom.tyBtnMagAIVPosSen2.bValue			:= p_tyDI.bMag2AIVInPosSen2;
	tyP0931MagConv2.tyCom.tyBtnMagOrientationChkSen1.bValue	:= p_tyDI.bMag2OrientChkSen1;
	tyP0931MagConv2.tyCom.tyBtnMagOrientationChkSen2.bValue	:= p_tyDI.bMag2OrientChkSen2;

	tyP0931MagConv2.tyCom.tyBtnFixedClampRS.bValue			:= p_tyDI.bMag2FixedClampRS;
	tyP0931MagConv2.tyCom.tyBtnFixedUnclampRS.bValue		:= p_tyDI.bMag2FixedUnclampRS;
	tyP0931MagConv2.tyCom.tyBtnRemoteClampRS.bValue			:= p_tyDI.bMag2RemoteClampRS;
	tyP0931MagConv2.tyCom.tyBtnRemoteUnclampRS.bValue		:= p_tyDI.bMag2RemoteUnclampRS;

	tyP0931MagConv2.tyCom.tyBtnSelUnclampRS.bValue			:= p_tyDI.bMag2SelUnClampRS;

	tyP0931MagConv2.tyCom.tyBtnCAB717Sen.bValue				:= p_tyDI.bMagConvCAB717MagSen2;
//	tyP0931MagConv2.tyCom.tyBtnHeightSen.bValue				:= p_tyDI.bMagConvHeightSen2;
	tyP0931MagConv2.tyCom.tyBtnMagSmallSen.bValue			:= p_tyDI.bMagConvSmallMagSen2;
	tyP0931MagConv2.tyCom.tyBtnMagLargeSen.bValue			:= p_tyDI.bMagConvLargeMagSen2;

	tyP0931MagConv2.tyCom.tyBtnMagDetectSen.bValue			:= p_tyDI.bMag2FixedClampSen;
//	tyP0931MagConv2.tyCom.tyBtnMagDetectSen.uiRtStat.0		:= NOT p_tyNtParamCurr.bProjFixClprMagDetectSenPrep;

	IF p_tyNtParamCurr.bMagAutoVerifyPrep = TRUE THEN
		tyP0931MagConv2.tyCom.tyBtnHeightSen.bValue			:= p_tyDI.bMagConvHeightSen2;
	ELSE
		tyP0931MagConv2.tyCom.tyBtnHeightSen.bValue			:= p_tyDI.bHighMagDetSen2;
	END_IF

	//Machine Bitmap
	IF p_tyNtParamCurr.eProjMag = ULMagDual AND p_tyNtParamCurr.bMagAutoVerifyPrep = FALSE THEN
		IF tyP0931MagConv2.tyFB.tyBtnFixedClamp.bRtCompl (*Bottom*)
			OR tyP0931MagConv2.tyDC.tyBtnFixedClamp.bRtCompl THEN

			tyP0931MagConv2.tyCom.tyBitmapMc.uiValueIdx	:= 109;

		ELSIF tyP0931MagConv2.tyFB.tyBtnFixedUnclamp.bRtCompl
			OR tyP0931MagConv2.tyDC.tyBtnFixedUnclamp.bRtCompl THEN

			tyP0931MagConv2.tyCom.tyBitmapMc.uiValueIdx	:= 108;

		ELSIF tyP0931MagConv2.tyFB.tyBtnRemoteClamp.bRtCompl (*Top*)
			OR tyP0931MagConv2.tyDC.tyBtnRemoteClamp.bRtCompl THEN

			tyP0931MagConv2.tyCom.tyBitmapMc.uiValueIdx	:= 113;

		ELSIF tyP0931MagConv2.tyFB.tyBtnRemoteUnclamp.bRtCompl
			OR tyP0931MagConv2.tyDC.tyBtnRemoteUnclamp.bRtCompl THEN

			tyP0931MagConv2.tyCom.tyBitmapMc.uiValueIdx	:= 112;

		ELSIF tyP0931MagConv2.tyFB.tyBtnEnt.bRtCompl OR tyP0931MagConv2.tyFB.tyBtnExit.bRtCompl OR tyP0931MagConv2.tyFB.tyBtnStop.bRtCompl
			OR tyP0931MagConv2.tyDC.tyBtnMagIn.bRtCompl OR tyP0931MagConv2.tyDC.tyBtnMagOut.bRtCompl OR tyP0931MagConv2.tyDC.tyBtnStop.bRtCompl THEN

			tyP0931MagConv2.tyCom.tyBitmapMc.uiValueIdx	:= 107;

		END_IF
	ELSIF p_tyNtParamCurr.bMagAutoVerifyPrep AND p_tyNtParamCurr.bProjMagAWPrep = FALSE THEN
		IF tyP0931MagConv2.tyFB.tyBtnFixedClamp.bRtCompl (*Bottom*)
			OR tyP0931MagConv2.tyDC.tyBtnFixedClamp.bRtCompl THEN

			tyP0931MagConv2.tyCom.tyBitmapMc.uiValueIdx	:= 23;

		ELSIF tyP0931MagConv2.tyFB.tyBtnFixedUnclamp.bRtCompl
			OR tyP0931MagConv2.tyDC.tyBtnFixedUnclamp.bRtCompl THEN

			tyP0931MagConv2.tyCom.tyBitmapMc.uiValueIdx	:= 24;

		ELSIF tyP0931MagConv2.tyFB.tyBtnRemoteClamp.bRtCompl (*Top*)
			OR tyP0931MagConv2.tyDC.tyBtnRemoteClamp.bRtCompl THEN

			tyP0931MagConv2.tyCom.tyBitmapMc.uiValueIdx	:= 18;

		ELSIF tyP0931MagConv2.tyFB.tyBtnRemoteUnclamp.bRtCompl
			OR tyP0931MagConv2.tyDC.tyBtnRemoteUnclamp.bRtCompl THEN

			tyP0931MagConv2.tyCom.tyBitmapMc.uiValueIdx	:= 17;

		ELSIF tyP0931MagConv2.tyFB.tyBtnSelClamp.bRtCompl
			OR tyP0931MagConv2.tyDC.tyBtnSelClamp.bRtCompl THEN

			tyP0931MagConv2.tyCom.tyBitmapMc.uiValueIdx	:= 29;

		ELSIF tyP0931MagConv2.tyFB.tyBtnSelUnclamp.bRtCompl
			OR tyP0931MagConv2.tyDC.tyBtnSelUnclamp.bRtCompl THEN

			tyP0931MagConv2.tyCom.tyBitmapMc.uiValueIdx	:= 30;

		ELSIF tyP0931MagConv2.tyFB.tyBtnEnt.bRtCompl OR tyP0931MagConv2.tyFB.tyBtnExit.bRtCompl OR tyP0931MagConv2.tyFB.tyBtnStop.bRtCompl
			OR tyP0931MagConv2.tyDC.tyBtnMagIn.bRtCompl OR tyP0931MagConv2.tyDC.tyBtnMagOut.bRtCompl OR tyP0931MagConv2.tyDC.tyBtnStop.bRtCompl THEN

			tyP0931MagConv2.tyCom.tyBitmapMc.uiValueIdx	:= 0;

		END_IF

	ELSIF p_tyNtParamCurr.eProjMag = ULMagTriple AND p_tyNtParamCurr.bMagAutoVerifyPrep AND p_tyNtParamCurr.bProjMagAWPrep AND p_tyNtParamCurr.bProjMotorizedPusherPrep = FALSE THEN
			IF tyP0931MagConv2.tyFB.tyBtnFixedClamp.bRtCompl (*Bottom*)
				OR tyP0931MagConv2.tyDC.tyBtnFixedClamp.bRtCompl THEN

				tyP0931MagConv2.tyCom.tyBitmapMc.uiValueIdx	:= 47;

			ELSIF tyP0931MagConv2.tyFB.tyBtnFixedUnclamp.bRtCompl
				OR tyP0931MagConv2.tyDC.tyBtnFixedUnclamp.bRtCompl THEN

				tyP0931MagConv2.tyCom.tyBitmapMc.uiValueIdx	:= 48;

			ELSIF tyP0931MagConv2.tyFB.tyBtnRemoteClamp.bRtCompl (*Top*)
				OR tyP0931MagConv2.tyDC.tyBtnRemoteClamp.bRtCompl THEN

				tyP0931MagConv2.tyCom.tyBitmapMc.uiValueIdx	:= 60;

			ELSIF tyP0931MagConv2.tyFB.tyBtnRemoteUnclamp.bRtCompl
				OR tyP0931MagConv2.tyDC.tyBtnRemoteUnclamp.bRtCompl THEN

				tyP0931MagConv2.tyCom.tyBitmapMc.uiValueIdx	:= 59;

			ELSIF tyP0931MagConv2.tyFB.tyBtnSelClamp.bRtCompl
				OR tyP0931MagConv2.tyDC.tyBtnSelClamp.bRtCompl THEN

				tyP0931MagConv2.tyCom.tyBitmapMc.uiValueIdx	:= 42;

			ELSIF tyP0931MagConv2.tyFB.tyBtnSelUnclamp.bRtCompl
				OR tyP0931MagConv2.tyDC.tyBtnSelUnclamp.bRtCompl THEN

				tyP0931MagConv2.tyCom.tyBitmapMc.uiValueIdx	:= 41;

			ELSIF tyP0931MagConv2.tyFB.tyBtnEnt.bRtCompl OR tyP0931MagConv2.tyFB.tyBtnExit.bRtCompl OR tyP0931MagConv2.tyFB.tyBtnStop.bRtCompl
				OR tyP0931MagConv2.tyDC.tyBtnMagIn.bRtCompl OR tyP0931MagConv2.tyDC.tyBtnMagOut.bRtCompl OR tyP0931MagConv2.tyDC.tyBtnStop.bRtCompl THEN

				tyP0931MagConv2.tyCom.tyBitmapMc.uiValueIdx	:= 3;

			END_IF

		ELSIF  p_tyNtParamCurr.eProjMag = ULMagTriple AND p_tyNtParamCurr.bMagAutoVerifyPrep = FALSE AND p_tyNtParamCurr.bProjMagAWPrep = FALSE AND p_tyNtParamCurr.bProjMotorizedPusherPrep THEN
			IF tyP0931MagConv2.tyFB.tyBtnFixedClamp.bRtCompl
				OR tyP0931MagConv2.tyDC.tyBtnFixedClamp.bRtCompl THEN
					IF p_tyNtParamCurr.bCurtainSenPrep THEN
						tyP0931MagConv2.tyCom.tyBitmapMc.uiValueIdx	:= 233;
					ELSE
						tyP0931MagConv2.tyCom.tyBitmapMc.uiValueIdx	:= 205;
					END_IF
			ELSIF tyP0931MagConv2.tyFB.tyBtnFixedUnclamp.bRtCompl
				OR tyP0931MagConv2.tyDC.tyBtnFixedUnclamp.bRtCompl THEN

					IF p_tyNtParamCurr.bCurtainSenPrep THEN
						tyP0931MagConv2.tyCom.tyBitmapMc.uiValueIdx	:= 233;
					ELSE
						tyP0931MagConv2.tyCom.tyBitmapMc.uiValueIdx	:= 204;
					END_IF

			ELSIF tyP0931MagConv2.tyFB.tyBtnRemoteClamp.bRtCompl
				OR tyP0931MagConv2.tyDC.tyBtnRemoteClamp.bRtCompl THEN

					IF p_tyNtParamCurr.bCurtainSenPrep THEN
						tyP0931MagConv2.tyCom.tyBitmapMc.uiValueIdx	:= 233;
					ELSE
						tyP0931MagConv2.tyCom.tyBitmapMc.uiValueIdx	:= 218;
					END_IF

			ELSIF tyP0931MagConv2.tyFB.tyBtnRemoteUnclamp.bRtCompl
				OR tyP0931MagConv2.tyDC.tyBtnRemoteUnclamp.bRtCompl THEN

					IF p_tyNtParamCurr.bCurtainSenPrep THEN
						tyP0931MagConv2.tyCom.tyBitmapMc.uiValueIdx	:= 233;
					ELSE
						tyP0931MagConv2.tyCom.tyBitmapMc.uiValueIdx	:= 217;
					END_IF

				//				ELSIF tyP0930MagConv2.tyFB.tyBtnSelClamp.bRtCompl
				//					OR tyP0930MagConv2.tyDC.tyBtnSelClamp.bRtCompl THEN
				//
				//					tyP0930MagConv2.tyCom.tyBitmapMc.uiValueIdx	:= 41;
				//
				//				ELSIF tyP0930MagConv2.tyFB.tyBtnSelUnclamp.bRtCompl
				//					OR tyP0930MagConv2.tyDC.tyBtnSelUnclamp.bRtCompl THEN
				//
				//					tyP0930MagConv1.tyCom.tyBitmapMc.uiValueIdx	:= 40;
				//
			ELSIF tyP0931MagConv2.tyFB.tyBtnEnt.bRtCompl OR tyP0931MagConv2.tyFB.tyBtnExit.bRtCompl OR tyP0931MagConv2.tyFB.tyBtnStop.bRtCompl
				OR tyP0931MagConv2.tyDC.tyBtnMagIn.bRtCompl OR tyP0931MagConv2.tyDC.tyBtnMagOut.bRtCompl OR tyP0931MagConv2.tyDC.tyBtnStop.bRtCompl THEN

				IF p_tyNtParamCurr.bCurtainSenPrep THEN
					tyP0931MagConv2.tyCom.tyBitmapMc.uiValueIdx	:= 234;
				ELSE
					tyP0931MagConv2.tyCom.tyBitmapMc.uiValueIdx	:= 203;
				END_IF

			END_IF
		ELSIF p_tyNtParamCurr.eProjMag = ULMagDual THEN
			IF tyP0931MagConv2.tyFB.tyBtnFixedClamp.bRtCompl (*Bottom*)
				OR tyP0931MagConv2.tyDC.tyBtnFixedClamp.bRtCompl THEN

				tyP0931MagConv2.tyCom.tyBitmapMc.uiValueIdx	:= 147;

			ELSIF tyP0931MagConv2.tyFB.tyBtnFixedUnclamp.bRtCompl
				OR tyP0931MagConv2.tyDC.tyBtnFixedUnclamp.bRtCompl THEN

				tyP0931MagConv2.tyCom.tyBitmapMc.uiValueIdx	:= 148;

			ELSIF tyP0931MagConv2.tyFB.tyBtnRemoteClamp.bRtCompl (*Top*)
				OR tyP0931MagConv2.tyDC.tyBtnRemoteClamp.bRtCompl THEN

				tyP0931MagConv2.tyCom.tyBitmapMc.uiValueIdx	:= 160;

			ELSIF tyP0931MagConv2.tyFB.tyBtnRemoteUnclamp.bRtCompl
				OR tyP0931MagConv2.tyDC.tyBtnRemoteUnclamp.bRtCompl THEN

				tyP0931MagConv2.tyCom.tyBitmapMc.uiValueIdx	:= 159;

			ELSIF tyP0931MagConv2.tyFB.tyBtnSelClamp.bRtCompl
				OR tyP0931MagConv2.tyDC.tyBtnSelClamp.bRtCompl THEN

				tyP0931MagConv2.tyCom.tyBitmapMc.uiValueIdx	:= 142;

			ELSIF tyP0931MagConv2.tyFB.tyBtnSelUnclamp.bRtCompl
				OR tyP0931MagConv2.tyDC.tyBtnSelUnclamp.bRtCompl THEN

				tyP0931MagConv2.tyCom.tyBitmapMc.uiValueIdx	:= 141;

			ELSIF tyP0931MagConv2.tyFB.tyBtnEnt.bRtCompl OR tyP0931MagConv2.tyFB.tyBtnExit.bRtCompl OR tyP0931MagConv2.tyFB.tyBtnStop.bRtCompl
				OR tyP0931MagConv2.tyDC.tyBtnMagIn.bRtCompl OR tyP0931MagConv2.tyDC.tyBtnMagOut.bRtCompl OR tyP0931MagConv2.tyDC.tyBtnStop.bRtCompl THEN

					tyP0931MagConv2.tyCom.tyBitmapMc.uiValueIdx	:= 103;

				END_IF
		END_IF

//	IF p_tyNtParamCurr.eProjMag = ULMagTriple AND p_tyNtParamCurr.bMagAutoVerifyPrep = FALSE THEN
//		IF tyP0931MagConv2.tyCom.tyBitmapMc.uiValueIdx < 100 THEN
//			tyP0931MagConv2.tyCom.tyBitmapMc.uiValueIdx	:= tyP0931MagConv2.tyCom.tyBitmapMc.uiValueIdx + 100;
//		END_IF
//	ELSIF p_tyNtParamCurr.eProjMag = ULMagTriple AND p_tyNtParamCurr.bMagAutoVerifyPrep = TRUE THEN
//		IF tyP0931MagConv2.tyCom.tyBitmapMc.uiValueIdx < 200 THEN
//			tyP0931MagConv2.tyCom.tyBitmapMc.uiValueIdx	:= tyP0931MagConv2.tyCom.tyBitmapMc.uiValueIdx + 200;
//		END_IF
//	END_IF

END_ACTION
```
